LIN {X 0,Y 298.79,Z 342.264,A -85,B 0,C 180,E1 -16386.754,E2 -16386.754} C_VEL
LIN {X 0,Y 298.673,Z 342.283,A -85,B 0,C 180,E1 -16389.481,E2 -16389.481} C_VEL
LIN {X 0,Y 298.544,Z 342.297,A -85,B 0,C 180,E1 -16393.616,E2 -16393.616} C_VEL
LIN {X 0,Y 298.541,Z 342.295,A -85,B 0,C 180,E1 -16396.409,E2 -16396.409} C_VEL
LIN {X 0,Y 298.503,Z 342.301,A -85,B 0,C 180,E1 -16399.655,E2 -16399.655} C_VEL
LIN {X 0,Y 298.416,Z 342.312,A -85,B 0,C 180,E1 -16403.601,E2 -16403.601} C_VEL
LIN {X 0,Y 298.4,Z 342.315,A -85,B 0,C 180,E1 -16406.583,E2 -16406.583} C_VEL
LIN {X 0,Y 298.386,Z 342.315,A -85,B 0,C 180,E1 -16409.645,E2 -16409.645} C_VEL
LIN {X 0,Y 298.386,Z 342.319,A -85,B 0,C 180,E1 -16412.802,E2 -16412.802} C_VEL
LIN {X 0,Y 298.435,Z 342.313,A -85,B 0,C 180,E1 -16416.807,E2 -16416.807} C_VEL
LIN {X 0,Y 298.342,Z 342.321,A -85,B 0,C 180,E1 -16421.08,E2 -16421.08} C_VEL
LIN {X 0,Y 298.35,Z 342.321,A -85,B 0,C 180,E1 -16425.036,E2 -16425.036} C_VEL
LIN {X 0,Y 298.428,Z 342.312,A -85,B 0,C 180,E1 -16426.927,E2 -16426.927} C_VEL
LIN {X 0,Y 298.392,Z 342.316,A -85,B 0,C 180,E1 -16431.009,E2 -16431.009} C_VEL
LIN {X 0,Y 298.515,Z 343.786,A -85,B 0,C 180,E1 -16433.175,E2 -16433.175} C_VEL
LIN {X 0,Y 298.505,Z 345.953,A -85,B 0,C 180,E1 -16435.595,E2 -16435.595} C_VEL
LIN {X 0,Y 298.24,Z 348.977,A -85,B 0,C 180,E1 -16438.774,E2 -16438.774} C_VEL
LIN {X 0,Y 297.975,Z 352.015,A -85,B 0,C 180,E1 -16441.855,E2 -16441.855} C_VEL
LIN {X 0,Y 297.704,Z 355.744,A -85,B 0,C 180,E1 -16445.475,E2 -16445.475} C_VEL
LIN {X 0,Y 301.735,Z 369.34,A -85,B 0,C 180,E1 -16446.473,E2 -16446.473} C_VEL
LIN {X 0,Y 304.492,Z 381.011,A -85,B 0,C 180,E1 -16447.514,E2 -16447.514} C_VEL
LIN {X 0,Y 306.309,Z 391.773,A -85,B 0,C 180,E1 -16448.64,E2 -16448.64} C_VEL
LIN {X 0,Y 306.628,Z 395.068,A -85,B 0,C 180,E1 -16449.016,E2 -16449.016} C_VEL
LIN {X 0,Y 305.081,Z 406.409,A -85,B 0,C 180,E1 -16450.312,E2 -16450.312} C_VEL
LIN {X 0,Y 303.763,Z 416.336,A -85,B 0,C 180,E1 -16451.753,E2 -16451.753} C_VEL
LIN {X 0,Y 302.259,Z 425.786,A -85,B 0,C 180,E1 -16453.452,E2 -16453.452} C_VEL
LIN {X 0,Y 300.578,Z 434.694,A -85,B 0,C 180,E1 -16455.443,E2 -16455.443} C_VEL
LIN {X 0,Y 299.354,Z 441.858,A -85,B 0,C 180,E1 -16457.458,E2 -16457.458} C_VEL
LIN {X 0,Y 298.473,Z 446.69,A -85,B 0,C 180,E1 -16459.143,E2 -16459.143} C_VEL
LIN {X 0,Y 297.683,Z 451.382,A -85,B 0,C 180,E1 -16461.173,E2 -16461.173} C_VEL
LIN {X 0,Y 297.207,Z 455.108,A -85,B 0,C 180,E1 -16463.3,E2 -16463.3} C_VEL
LIN {X 0,Y 296.959,Z 456.824,A -85,B 0,C 180,E1 -16464.569,E2 -16464.569} C_VEL
LIN {X 0,Y 296.811,Z 458.217,A -85,B 0,C 180,E1 -16465.927,E2 -16465.927} C_VEL
LIN {X 0,Y 296.546,Z 459.821,A -85,B 0,C 180,E1 -16468.643,E2 -16468.643} C_VEL
LIN {X 0,Y 296.529,Z 460.051,A -85,B 0,C 180,E1 -16470.001,E2 -16470.001} C_VEL
LIN {X 0,Y 296.546,Z 459.859,A -85,B 0,C 180,E1 -16471.359,E2 -16471.359} C_VEL
LIN {X 0,Y 296.788,Z 458.304,A -85,B 0,C 180,E1 -16474.074,E2 -16474.074} C_VEL
LIN {X 0,Y 296.96,Z 456.948,A -85,B 0,C 180,E1 -16475.433,E2 -16475.433} C_VEL
LIN {X 0,Y 297.357,Z 454.082,A -85,B 0,C 180,E1 -16477.47,E2 -16477.47} C_VEL
LIN {X 0,Y 297.855,Z 450.199,A -85,B 0,C 180,E1 -16479.507,E2 -16479.507} C_VEL
LIN {X 0,Y 298.758,Z 445.181,A -85,B 0,C 180,E1 -16481.535,E2 -16481.535} C_VEL
LIN {X 0,Y 299.867,Z 438.863,A -85,B 0,C 180,E1 -16483.555,E2 -16483.555} C_VEL
LIN {X 0,Y 301.325,Z 430.953,A -85,B 0,C 180,E1 -16485.559,E2 -16485.559} C_VEL
LIN {X 0,Y 303.025,Z 421.112,A -85,B 0,C 180,E1 -16487.548,E2 -16487.548} C_VEL
LIN {X 0,Y 304.471,Z 410.784,A -85,B 0,C 180,E1 -16489.204,E2 -16489.204} C_VEL
LIN {X 0,Y 306.134,Z 399.125,A -85,B 0,C 180,E1 -16490.669,E2 -16490.669} C_VEL
LIN {X 0,Y 306.659,Z 394.489,A -85,B 0,C 180,E1 -16491.159,E2 -16491.159} C_VEL
LIN {X 0,Y 304.975,Z 383.491,A -85,B 0,C 180,E1 -16492.36,E2 -16492.36} C_VEL
LIN {X 0,Y 302.381,Z 371.646,A -85,B 0,C 180,E1 -16493.45,E2 -16493.45} C_VEL
LIN {X 0,Y 298.518,Z 358.662,A -85,B 0,C 180,E1 -16494.449,E2 -16494.449} C_VEL
LIN {X 0,Y 297.688,Z 355.729,A -85,B 0,C 180,E1 -16494.66,E2 -16494.66} C_VEL
LIN {X 0,Y 297.944,Z 352.136,A -85,B 0,C 180,E1 -16498.149,E2 -16498.149} C_VEL
LIN {X 0,Y 298.325,Z 348.377,A -85,B 0,C 180,E1 -16501.994,E2 -16501.994} C_VEL
LIN {X 0,Y 298.503,Z 345.997,A -85,B 0,C 180,E1 -16504.508,E2 -16504.508} C_VEL
LIN {X 0,Y 298.455,Z 343.087,A -85,B 0,C 180,E1 -16507.752,E2 -16507.752} C_VEL
LIN {X 0,Y 298.388,Z 342.318,A -85,B 0,C 180,E1 -16508.99,E2 -16508.99} C_VEL
LIN {X 0,Y 298.399,Z 342.317,A -85,B 0,C 180,E1 -16513.103,E2 -16513.103} C_VEL
LIN {X 0,Y 298.369,Z 342.319,A -85,B 0,C 180,E1 -16516.914,E2 -16516.914} C_VEL
LIN {X 0,Y 298.353,Z 342.32,A -85,B 0,C 180,E1 -16521.018,E2 -16521.018} C_VEL
LIN {X 0,Y 298.415,Z 342.312,A -85,B 0,C 180,E1 -16523.929,E2 -16523.929} C_VEL
LIN {X 0,Y 298.391,Z 342.318,A -85,B 0,C 180,E1 -16527.199,E2 -16527.199} C_VEL
LIN {X 0,Y 298.4,Z 342.314,A -85,B 0,C 180,E1 -16530.625,E2 -16530.625} C_VEL
LIN {X 0,Y 298.437,Z 342.31,A -85,B 0,C 180,E1 -16534.92,E2 -16534.92} C_VEL
LIN {X 0,Y 298.437,Z 342.31,A -85,B 0,C 180,E1 -16539.314,E2 -16539.314} C_VEL
LIN {X 0,Y 298.536,Z 342.296,A -85,B 0,C 180,E1 -16542.179,E2 -16542.179} C_VEL
LIN {X 0,Y 298.562,Z 342.293,A -85,B 0,C 180,E1 -16545.382,E2 -16545.382} C_VEL
LIN {X 0,Y 298.591,Z 342.29,A -85,B 0,C 180,E1 -16549.146,E2 -16549.146} C_VEL
LIN {X 0,Y 298.755,Z 342.269,A -85,B 0,C 180,E1 -16551.248,E2 -16551.248} C_VEL
LIN {X 0,Y 298.04,Z 342.361,A -85,B 0,C 180,E1 -16552.372,E2 -16552.372} C_VEL
LIN {X 0,Y 295.081,Z 342.728,A -85,B 0,C 180,E1 -16554.2,E2 -16554.2} C_VEL
LIN {X 0,Y 292.68,Z 343.025,A -85,B 0,C 180,E1 -16555.684,E2 -16555.684} C_VEL
LIN {X 0,Y 291.784,Z 343.139,A -85,B 0,C 180,E1 -16556.835,E2 -16556.835} C_VEL
LIN {X 0,Y 291.782,Z 343.137,A -85,B 0,C 180,E1 -16557.224,E2 -16557.224} C_VEL
LIN {X 0,Y 291.915,Z 343.123,A -85,B 0,C 180,E1 -16560,E2 -16560} C_VEL
LIN {X 0,Y 291.785,Z 343.138,A -85,B 0,C 180,E1 -16562.761,E2 -16562.761} C_VEL
LIN {X 0,Y 291.733,Z 343.144,A -85,B 0,C 180,E1 -16566.918,E2 -16566.918} C_VEL
LIN {X 0,Y 291.573,Z 343.166,A -85,B 0,C 180,E1 -16569.714,E2 -16569.714} C_VEL
LIN {X 0,Y 291.519,Z 343.175,A -85,B 0,C 180,E1 -16573.95,E2 -16573.95} C_VEL
LIN {X 0,Y 291.485,Z 343.175,A -85,B 0,C 180,E1 -16576.818,E2 -16576.818} C_VEL
LIN {X 0,Y 291.449,Z 343.183,A -85,B 0,C 180,E1 -16579.875,E2 -16579.875} C_VEL
LIN {X 0,Y 291.361,Z 343.191,A -85,B 0,C 180,E1 -16584.209,E2 -16584.209} C_VEL
LIN {X 0,Y 291.351,Z 343.194,A -85,B 0,C 180,E1 -16587.279,E2 -16587.279} C_VEL
LIN {X 0,Y 291.316,Z 343.197,A -85,B 0,C 180,E1 -16590.439,E2 -16590.439} C_VEL
LIN {X 0,Y 291.342,Z 343.197,A -85,B 0,C 180,E1 -16593.699,E2 -16593.699} C_VEL
LIN {X 0,Y 291.358,Z 343.195,A -85,B 0,C 180,E1 -16597.25,E2 -16597.25} C_VEL
LIN {X 0,Y 291.298,Z 343.198,A -85,B 0,C 180,E1 -16600.648,E2 -16600.648} C_VEL
LIN {X 0,Y 291.369,Z 343.359,A -85,B 0,C 180,E1 -16602.483,E2 -16602.483} C_VEL
LIN {X 0,Y 292.046,Z 347.294,A -85,B 0,C 180,E1 -16606.215,E2 -16606.215} C_VEL
LIN {X 0,Y 292.85,Z 351.787,A -85,B 0,C 180,E1 -16610.171,E2 -16610.171} C_VEL
LIN {X 0,Y 293.099,Z 355.448,A -85,B 0,C 180,E1 -16613.169,E2 -16613.169} C_VEL
LIN {X 0,Y 292.963,Z 358.663,A -85,B 0,C 180,E1 -16615.685,E2 -16615.685} C_VEL
LIN {X 0,Y 292.107,Z 364.486,A -85,B 0,C 180,E1 -16620.014,E2 -16620.014} C_VEL
LIN {X 0,Y 291.474,Z 368.769,A -85,B 0,C 180,E1 -16623.144,E2 -16623.144} C_VEL
LIN {X 0,Y 291.178,Z 371.049,A -85,B 0,C 180,E1 -16624.786,E2 -16624.786} C_VEL
LIN {X 0,Y 294.511,Z 384.98,A -85,B 0,C 180,E1 -16625.735,E2 -16625.735} C_VEL
LIN {X 0,Y 296.709,Z 397.246,A -85,B 0,C 180,E1 -16626.775,E2 -16626.775} C_VEL
LIN {X 0,Y 298.098,Z 409.454,A -85,B 0,C 180,E1 -16628.021,E2 -16628.021} C_VEL
LIN {X 0,Y 298.565,Z 417.315,A -85,B 0,C 180,E1 -16628.963,E2 -16628.963} C_VEL
LIN {X 0,Y 296.81,Z 428.854,A -85,B 0,C 180,E1 -16630.46,E2 -16630.46} C_VEL
LIN {X 0,Y 295.151,Z 439.157,A -85,B 0,C 180,E1 -16632.167,E2 -16632.167} C_VEL
LIN {X 0,Y 293.594,Z 448.125,A -85,B 0,C 180,E1 -16634.021,E2 -16634.021} C_VEL
LIN {X 0,Y 292.189,Z 456.149,A -85,B 0,C 180,E1 -16636.082,E2 -16636.082} C_VEL
LIN {X 0,Y 291.085,Z 462.584,A -85,B 0,C 180,E1 -16638.157,E2 -16638.157} C_VEL
LIN {X 0,Y 290.314,Z 467.698,A -85,B 0,C 180,E1 -16640.243,E2 -16640.243} C_VEL
LIN {X 0,Y 289.82,Z 471.673,A -85,B 0,C 180,E1 -16642.335,E2 -16642.335} C_VEL
LIN {X 0,Y 289.517,Z 474.61,A -85,B 0,C 180,E1 -16644.427,E2 -16644.427} C_VEL
LIN {X 0,Y 289.451,Z 476.01,A -85,B 0,C 180,E1 -16645.822,E2 -16645.822} C_VEL
LIN {X 0,Y 289.442,Z 477.01,A -85,B 0,C 180,E1 -16647.216,E2 -16647.216} C_VEL
LIN {X 0,Y 289.403,Z 477.619,A -85,B 0,C 180,E1 -16648.608,E2 -16648.608} C_VEL
LIN {X 0,Y 289.406,Z 477.834,A -85,B 0,C 180,E1 -16649.999,E2 -16649.999} C_VEL
LIN {X 0,Y 289.403,Z 477.615,A -85,B 0,C 180,E1 -16651.391,E2 -16651.391} C_VEL
LIN {X 0,Y 289.441,Z 477.004,A -85,B 0,C 180,E1 -16652.783,E2 -16652.783} C_VEL
LIN {X 0,Y 289.45,Z 476.002,A -85,B 0,C 180,E1 -16654.177,E2 -16654.177} C_VEL
LIN {X 0,Y 289.517,Z 474.598,A -85,B 0,C 180,E1 -16655.571,E2 -16655.571} C_VEL
LIN {X 0,Y 289.812,Z 471.652,A -85,B 0,C 180,E1 -16657.664,E2 -16657.664} C_VEL
LIN {X 0,Y 290.314,Z 467.667,A -85,B 0,C 180,E1 -16659.755,E2 -16659.755} C_VEL
LIN {X 0,Y 291.204,Z 461.543,A -85,B 0,C 180,E1 -16662.19,E2 -16662.19} C_VEL
LIN {X 0,Y 292.408,Z 454.86,A -85,B 0,C 180,E1 -16664.261,E2 -16664.261} C_VEL
LIN {X 0,Y 293.894,Z 446.57,A -85,B 0,C 180,E1 -16666.318,E2 -16666.318} C_VEL
LIN {X 0,Y 295.282,Z 438.07,A -85,B 0,C 180,E1 -16668.023,E2 -16668.023} C_VEL
LIN {X 0,Y 296.951,Z 427.571,A -85,B 0,C 180,E1 -16669.709,E2 -16669.709} C_VEL
LIN {X 0,Y 298.54,Z 417.189,A -85,B 0,C 180,E1 -16671.038,E2 -16671.038} C_VEL
LIN {X 0,Y 297.747,Z 405.797,A -85,B 0,C 180,E1 -16672.363,E2 -16672.363} C_VEL
LIN {X 0,Y 296.101,Z 393.226,A -85,B 0,C 180,E1 -16673.567,E2 -16673.567} C_VEL
LIN {X 0,Y 293.606,Z 380.807,A -85,B 0,C 180,E1 -16674.55,E2 -16674.55} C_VEL
LIN {X 0,Y 291.195,Z 371.057,A -85,B 0,C 180,E1 -16675.187,E2 -16675.187} C_VEL
LIN {X 0,Y 291.859,Z 366.099,A -85,B 0,C 180,E1 -16678.789,E2 -16678.789} C_VEL
LIN {X 0,Y 292.669,Z 360.646,A -85,B 0,C 180,E1 -16682.81,E2 -16682.81} C_VEL
LIN {X 0,Y 293.112,Z 357.233,A -85,B 0,C 180,E1 -16685.39,E2 -16685.39} C_VEL
LIN {X 0,Y 293.05,Z 353.256,A -85,B 0,C 180,E1 -16688.573,E2 -16688.573} C_VEL
LIN {X 0,Y 292.495,Z 349.393,A -85,B 0,C 180,E1 -16691.853,E2 -16691.853} C_VEL
LIN {X 0,Y 291.72,Z 345.229,A -85,B 0,C 180,E1 -16695.681,E2 -16695.681} C_VEL
LIN {X 0,Y 291.343,Z 343.196,A -85,B 0,C 180,E1 -16697.767,E2 -16697.767} C_VEL
LIN {X 0,Y 291.328,Z 343.199,A -85,B 0,C 180,E1 -16701.154,E2 -16701.154} C_VEL
LIN {X 0,Y 291.349,Z 343.196,A -85,B 0,C 180,E1 -16704.624,E2 -16704.624} C_VEL
LIN {X 0,Y 291.359,Z 343.192,A -85,B 0,C 180,E1 -16707.949,E2 -16707.949} C_VEL
LIN {X 0,Y 291.336,Z 343.195,A -85,B 0,C 180,E1 -16711.153,E2 -16711.153} C_VEL
LIN {X 0,Y 291.354,Z 343.195,A -85,B 0,C 180,E1 -16714.266,E2 -16714.266} C_VEL
LIN {X 0,Y 291.365,Z 343.19,A -85,B 0,C 180,E1 -16717.298,E2 -16717.298} C_VEL
LIN {X 0,Y 291.451,Z 343.182,A -85,B 0,C 180,E1 -16720.27,E2 -16720.27} C_VEL
LIN {X 0,Y 291.533,Z 343.17,A -85,B 0,C 180,E1 -16724.634,E2 -16724.634} C_VEL
LIN {X 0,Y 291.528,Z 343.168,A -85,B 0,C 180,E1 -16728.88,E2 -16728.88} C_VEL
LIN {X 0,Y 291.702,Z 343.15,A -85,B 0,C 180,E1 -16731.688,E2 -16731.688} C_VEL
LIN {X 0,Y 291.625,Z 343.157,A -85,B 0,C 180,E1 -16734.468,E2 -16734.468} C_VEL
LIN {X 0,Y 291.876,Z 343.125,A -85,B 0,C 180,E1 -16738.62,E2 -16738.62} C_VEL
LIN {X 0,Y 291.876,Z 343.128,A -85,B 0,C 180,E1 -16741.38,E2 -16741.38} C_VEL
LIN {X 0,Y 291.739,Z 343.143,A -85,B 0,C 180,E1 -16746.918,E2 -16746.918} C_VEL
LIN {X 0,Y 291.621,Z 343.16,A -85,B 0,C 180,E1 -16749.712,E2 -16749.712} C_VEL
LIN {X 0,Y 291.514,Z 343.17,A -85,B 0,C 180,E1 -16753.951,E2 -16753.951} C_VEL
LIN {X 0,Y 291.479,Z 343.176,A -85,B 0,C 180,E1 -16756.818,E2 -16756.818} C_VEL
LIN {X 0,Y 291.444,Z 343.179,A -85,B 0,C 180,E1 -16759.875,E2 -16759.875} C_VEL
LIN {X 0,Y 291.356,Z 343.19,A -85,B 0,C 180,E1 -16764.209,E2 -16764.209} C_VEL
LIN {X 0,Y 291.346,Z 343.194,A -85,B 0,C 180,E1 -16767.279,E2 -16767.279} C_VEL
LIN {X 0,Y 291.312,Z 343.198,A -85,B 0,C 180,E1 -16770.44,E2 -16770.44} C_VEL
LIN {X 0,Y 291.337,Z 343.193,A -85,B 0,C 180,E1 -16773.7,E2 -16773.7} C_VEL
LIN {X 0,Y 291.362,Z 343.191,A -85,B 0,C 180,E1 -16777.253,E2 -16777.253} C_VEL
LIN {X 0,Y 291.294,Z 343.201,A -85,B 0,C 180,E1 -16780.649,E2 -16780.649} C_VEL
LIN {X 0,Y 291.278,Z 343.204,A -85,B 0,C 180,E1 -16784.405,E2 -16784.405} C_VEL
LIN {X 0,Y 291.352,Z 343.195,A -85,B 0,C 180,E1 -16788.399,E2 -16788.399} C_VEL
LIN {X 0,Y 291.335,Z 343.195,A -85,B 0,C 180,E1 -16791.157,E2 -16791.157} C_VEL
LIN {X 0,Y 291.471,Z 344.663,A -85,B 0,C 180,E1 -16792.931,E2 -16792.931} C_VEL
LIN {X 0,Y 291.403,Z 347.671,A -85,B 0,C 180,E1 -16796.311,E2 -16796.311} C_VEL
LIN {X 0,Y 291.113,Z 350.699,A -85,B 0,C 180,E1 -16799.539,E2 -16799.539} C_VEL
LIN {X 0,Y 290.796,Z 354.517,A -85,B 0,C 180,E1 -16803.409,E2 -16803.409} C_VEL
LIN {X 0,Y 290.677,Z 355.97,A -85,B 0,C 180,E1 -16804.836,E2 -16804.836} C_VEL
LIN {X 0,Y 294.851,Z 369.828,A -85,B 0,C 180,E1 -16805.905,E2 -16805.905} C_VEL
LIN {X 0,Y 297.743,Z 381.66,A -85,B 0,C 180,E1 -16807.009,E2 -16807.009} C_VEL
LIN {X 0,Y 299.48,Z 392.003,A -85,B 0,C 180,E1 -16808.128,E2 -16808.128} C_VEL
LIN {X 0,Y 299.824,Z 396.866,A -85,B 0,C 180,E1 -16808.696,E2 -16808.696} C_VEL
LIN {X 0,Y 298.24,Z 407.907,A -85,B 0,C 180,E1 -16810.021,E2 -16810.021} C_VEL
LIN {X 0,Y 296.925,Z 417.177,A -85,B 0,C 180,E1 -16811.427,E2 -16811.427} C_VEL
LIN {X 0,Y 295.447,Z 426.004,A -85,B 0,C 180,E1 -16813.059,E2 -16813.059} C_VEL
LIN {X 0,Y 293.718,Z 434.912,A -85,B 0,C 180,E1 -16815.096,E2 -16815.096} C_VEL
LIN {X 0,Y 292.423,Z 442.076,A -85,B 0,C 180,E1 -16817.156,E2 -16817.156} C_VEL
LIN {X 0,Y 291.503,Z 446.907,A -85,B 0,C 180,E1 -16818.88,E2 -16818.88} C_VEL
LIN {X 0,Y 290.662,Z 451.599,A -85,B 0,C 180,E1 -16820.958,E2 -16820.958} C_VEL
LIN {X 0,Y 290.119,Z 455.604,A -85,B 0,C 180,E1 -16823.32,E2 -16823.32} C_VEL
LIN {X 0,Y 289.73,Z 458.433,A -85,B 0,C 180,E1 -16825.828,E2 -16825.828} C_VEL
LIN {X 0,Y 289.467,Z 460.036,A -85,B 0,C 180,E1 -16828.609,E2 -16828.609} C_VEL
LIN {X 0,Y 289.446,Z 460.266,A -85,B 0,C 180,E1 -16830.001,E2 -16830.001} C_VEL
LIN {X 0,Y 289.467,Z 460.073,A -85,B 0,C 180,E1 -16831.392,E2 -16831.392} C_VEL
LIN {X 0,Y 289.709,Z 458.519,A -85,B 0,C 180,E1 -16834.174,E2 -16834.174} C_VEL
LIN {X 0,Y 290.119,Z 455.759,A -85,B 0,C 180,E1 -16836.679,E2 -16836.679} C_VEL
LIN {X 0,Y 290.628,Z 451.826,A -85,B 0,C 180,E1 -16839.044,E2 -16839.044} C_VEL
LIN {X 0,Y 291.469,Z 447.193,A -85,B 0,C 180,E1 -16841.122,E2 -16841.122} C_VEL
LIN {X 0,Y 292.784,Z 440.208,A -85,B 0,C 180,E1 -16843.535,E2 -16843.535} C_VEL
LIN {X 0,Y 294.202,Z 432.635,A -85,B 0,C 180,E1 -16845.59,E2 -16845.59} C_VEL
LIN {X 0,Y 295.669,Z 424.872,A -85,B 0,C 180,E1 -16847.285,E2 -16847.285} C_VEL
LIN {X 0,Y 297.171,Z 414.978,A -85,B 0,C 180,E1 -16849.046,E2 -16849.046} C_VEL
LIN {X 0,Y 298.693,Z 404.861,A -85,B 0,C 180,E1 -16850.487,E2 -16850.487} C_VEL
LIN {X 0,Y 299.887,Z 396.275,A -85,B 0,C 180,E1 -16851.48,E2 -16851.48} C_VEL
LIN {X 0,Y 298.597,Z 386.445,A -85,B 0,C 180,E1 -16852.61,E2 -16852.61} C_VEL
LIN {X 0,Y 296.355,Z 375.616,A -85,B 0,C 180,E1 -16853.695,E2 -16853.695} C_VEL
LIN {X 0,Y 293.032,Z 363.689,A -85,B 0,C 180,E1 -16854.718,E2 -16854.718} C_VEL
LIN {X 0,Y 290.678,Z 355.979,A -85,B 0,C 180,E1 -16855.275,E2 -16855.275} C_VEL
LIN {X 0,Y 291.081,Z 351.622,A -85,B 0,C 180,E1 -16859.633,E2 -16859.633} C_VEL
LIN {X 0,Y 291.336,Z 349.015,A -85,B 0,C 180,E1 -16862.401,E2 -16862.401} C_VEL
LIN {X 0,Y 291.493,Z 346.287,A -85,B 0,C 180,E1 -16865.355,E2 -16865.355} C_VEL
LIN {X 0,Y 291.489,Z 344.587,A -85,B 0,C 180,E1 -16867.283,E2 -16867.283} C_VEL
LIN {X 0,Y 291.343,Z 343.282,A -85,B 0,C 180,E1 -16868.843,E2 -16868.843} C_VEL
LIN {X 0,Y 291.32,Z 343.198,A -85,B 0,C 180,E1 -16872.492,E2 -16872.492} C_VEL
LIN {X 0,Y 291.288,Z 343.201,A -85,B 0,C 180,E1 -16876.37,E2 -16876.37} C_VEL
LIN {X 0,Y 291.311,Z 343.196,A -85,B 0,C 180,E1 -16880.535,E2 -16880.535} C_VEL
LIN {X 0,Y 291.397,Z 343.187,A -85,B 0,C 180,E1 -16882.918,E2 -16882.918} C_VEL
LIN {X 0,Y 291.343,Z 343.192,A -85,B 0,C 180,E1 -16886.301,E2 -16886.301} C_VEL
LIN {X 0,Y 291.363,Z 343.189,A -85,B 0,C 180,E1 -16890.268,E2 -16890.268} C_VEL
LIN {X 0,Y 291.357,Z 343.19,A -85,B 0,C 180,E1 -16894.266,E2 -16894.266} C_VEL
LIN {X 0,Y 291.37,Z 343.19,A -85,B 0,C 180,E1 -16897.298,E2 -16897.298} C_VEL
LIN {X 0,Y 291.457,Z 343.178,A -85,B 0,C 180,E1 -16900.27,E2 -16900.27} C_VEL
LIN {X 0,Y 291.554,Z 343.169,A -85,B 0,C 180,E1 -16904.623,E2 -16904.623} C_VEL
LIN {X 0,Y 291.534,Z 343.171,A -85,B 0,C 180,E1 -16908.88,E2 -16908.88} C_VEL
LIN {X 0,Y 291.708,Z 343.146,A -85,B 0,C 180,E1 -16911.688,E2 -16911.688} C_VEL
LIN {X 0,Y 291.628,Z 343.161,A -85,B 0,C 180,E1 -16914.468,E2 -16914.468} C_VEL
LIN {X 0,Y 291.782,Z 343.137,A -85,B 0,C 180,E1 -16917.224,E2 -16917.224} C_VEL
LIN {X 0,Y 291.317,Z 343.201,A -85,B 0,C 180,E1 -16918.377,E2 -16918.377} C_VEL
LIN {X 0,Y 289.82,Z 343.389,A -85,B 0,C 180,E1 -16919.509,E2 -16919.509} C_VEL
LIN {X 0,Y 285.991,Z 343.861,A -85,B 0,C 180,E1 -16921.778,E2 -16921.778} C_VEL
LIN {X 0,Y 284.782,Z 344.01,A -85,B 0,C 180,E1 -16922.96,E2 -16922.96} C_VEL
LIN {X 0,Y 284.63,Z 344.028,A -85,B 0,C 180,E1 -16923.362,E2 -16923.362} C_VEL
LIN {X 0,Y 284.685,Z 344.022,A -85,B 0,C 180,E1 -16927.09,E2 -16927.09} C_VEL
LIN {X 0,Y 284.517,Z 344.047,A -85,B 0,C 180,E1 -16929.957,E2 -16929.957} C_VEL
LIN {X 0,Y 284.476,Z 344.051,A -85,B 0,C 180,E1 -16934.303,E2 -16934.303} C_VEL
LIN {X 0,Y 284.423,Z 344.056,A -85,B 0,C 180,E1 -16937.248,E2 -16937.248} C_VEL
LIN {X 0,Y 284.376,Z 344.062,A -85,B 0,C 180,E1 -16940.242,E2 -16940.242} C_VEL
LIN {X 0,Y 284.321,Z 344.07,A -85,B 0,C 180,E1 -16943.854,E2 -16943.854} C_VEL
LIN {X 0,Y 284.281,Z 344.075,A -85,B 0,C 180,E1 -16948.016,E2 -16948.016} C_VEL
LIN {X 0,Y 284.283,Z 344.076,A -85,B 0,C 180,E1 -16951.276,E2 -16951.276} C_VEL
LIN {X 0,Y 284.335,Z 344.07,A -85,B 0,C 180,E1 -16955.347,E2 -16955.347} C_VEL
LIN {X 0,Y 284.297,Z 344.072,A -85,B 0,C 180,E1 -16958.172,E2 -16958.172} C_VEL
LIN {X 0,Y 284.277,Z 344.153,A -85,B 0,C 180,E1 -16961.875,E2 -16961.875} C_VEL
LIN {X 0,Y 284.955,Z 348.026,A -85,B 0,C 180,E1 -16965.663,E2 -16965.663} C_VEL
LIN {X 0,Y 285.776,Z 352.392,A -85,B 0,C 180,E1 -16969.674,E2 -16969.674} C_VEL
LIN {X 0,Y 286.075,Z 356.323,A -85,B 0,C 180,E1 -16972.995,E2 -16972.995} C_VEL
LIN {X 0,Y 285.965,Z 359.535,A -85,B 0,C 180,E1 -16975.58,E2 -16975.58} C_VEL
LIN {X 0,Y 285.134,Z 364.816,A -85,B 0,C 180,E1 -16979.619,E2 -16979.619} C_VEL
LIN {X 0,Y 284.309,Z 370.096,A -85,B 0,C 180,E1 -16983.58,E2 -16983.58} C_VEL
LIN {X 0,Y 284.224,Z 370.828,A -85,B 0,C 180,E1 -16984.125,E2 -16984.125} C_VEL
LIN {X 0,Y 287.574,Z 384.322,A -85,B 0,C 180,E1 -16985.083,E2 -16985.083} C_VEL
LIN {X 0,Y 289.892,Z 397.148,A -85,B 0,C 180,E1 -16986.205,E2 -16986.205} C_VEL
LIN {X 0,Y 291.273,Z 409.236,A -85,B 0,C 180,E1 -16987.478,E2 -16987.478} C_VEL
LIN {X 0,Y 291.737,Z 418.533,A -85,B 0,C 180,E1 -16988.631,E2 -16988.631} C_VEL
LIN {X 0,Y 289.924,Z 429.774,A -85,B 0,C 180,E1 -16990.161,E2 -16990.161} C_VEL
LIN {X 0,Y 288.306,Z 439.314,A -85,B 0,C 180,E1 -16991.805,E2 -16991.805} C_VEL
LIN {X 0,Y 286.757,Z 447.911,A -85,B 0,C 180,E1 -16993.629,E2 -16993.629} C_VEL
LIN {X 0,Y 285.269,Z 455.934,A -85,B 0,C 180,E1 -16995.737,E2 -16995.737} C_VEL
LIN {X 0,Y 284.091,Z 462.368,A -85,B 0,C 180,E1 -16997.861,E2 -16997.861} C_VEL
LIN {X 0,Y 283.276,Z 467.482,A -85,B 0,C 180,E1 -16999.998,E2 -16999.998} C_VEL
LIN {X 0,Y 282.754,Z 471.457,A -85,B 0,C 180,E1 -17002.142,E2 -17002.142} C_VEL
LIN {X 0,Y 282.411,Z 474.64,A -85,B 0,C 180,E1 -17004.521,E2 -17004.521} C_VEL
LIN {X 0,Y 282.35,Z 476.795,A -85,B 0,C 180,E1 -17007.146,E2 -17007.146} C_VEL
LIN {X 0,Y 282.327,Z 477.404,A -85,B 0,C 180,E1 -17008.573,E2 -17008.573} C_VEL
LIN {X 0,Y 282.328,Z 477.62,A -85,B 0,C 180,E1 -17009.999,E2 -17009.999} C_VEL
LIN {X 0,Y 282.327,Z 477.4,A -85,B 0,C 180,E1 -17011.426,E2 -17011.426} C_VEL
LIN {X 0,Y 282.349,Z 476.788,A -85,B 0,C 180,E1 -17012.853,E2 -17012.853} C_VEL
LIN {X 0,Y 282.41,Z 474.628,A -85,B 0,C 180,E1 -17015.477,E2 -17015.477} C_VEL
LIN {X 0,Y 282.747,Z 471.435,A -85,B 0,C 180,E1 -17017.857,E2 -17017.857} C_VEL
LIN {X 0,Y 283.276,Z 467.449,A -85,B 0,C 180,E1 -17020,E2 -17020} C_VEL
LIN {X 0,Y 284.229,Z 461.325,A -85,B 0,C 180,E1 -17022.494,E2 -17022.494} C_VEL
LIN {X 0,Y 285.506,Z 454.641,A -85,B 0,C 180,E1 -17024.614,E2 -17024.614} C_VEL
LIN {X 0,Y 287.075,Z 446.352,A -85,B 0,C 180,E1 -17026.717,E2 -17026.717} C_VEL
LIN {X 0,Y 288.502,Z 437.85,A -85,B 0,C 180,E1 -17028.461,E2 -17028.461} C_VEL
LIN {X 0,Y 290.26,Z 427.352,A -85,B 0,C 180,E1 -17030.183,E2 -17030.183} C_VEL
LIN {X 0,Y 291.727,Z 418.398,A -85,B 0,C 180,E1 -17031.368,E2 -17031.368} C_VEL
LIN {X 0,Y 291.061,Z 407.28,A -85,B 0,C 180,E1 -17032.726,E2 -17032.726} C_VEL
LIN {X 0,Y 289.483,Z 394.534,A -85,B 0,C 180,E1 -17034.026,E2 -17034.026} C_VEL
LIN {X 0,Y 286.949,Z 381.735,A -85,B 0,C 180,E1 -17035.097,E2 -17035.097} C_VEL
LIN {X 0,Y 284.226,Z 370.799,A -85,B 0,C 180,E1 -17035.875,E2 -17035.875} C_VEL
LIN {X 0,Y 284.942,Z 365.886,A -85,B 0,C 180,E1 -17039.556,E2 -17039.556} C_VEL
LIN {X 0,Y 285.713,Z 361.03,A -85,B 0,C 180,E1 -17043.245,E2 -17043.245} C_VEL
LIN {X 0,Y 286.076,Z 357.364,A -85,B 0,C 180,E1 -17046.127,E2 -17046.127} C_VEL
LIN {X 0,Y 286.066,Z 354.879,A -85,B 0,C 180,E1 -17048.171,E2 -17048.171} C_VEL
LIN {X 0,Y 285.808,Z 352.343,A -85,B 0,C 180,E1 -17050.333,E2 -17050.333} C_VEL
LIN {X 0,Y 285.014,Z 347.953,A -85,B 0,C 180,E1 -17054.349,E2 -17054.349} C_VEL
LIN {X 0,Y 284.272,Z 344.077,A -85,B 0,C 180,E1 -17058.243,E2 -17058.243} C_VEL
LIN {X 0,Y 284.303,Z 344.072,A -85,B 0,C 180,E1 -17062.281,E2 -17062.281} C_VEL
LIN {X 0,Y 284.301,Z 344.071,A -85,B 0,C 180,E1 -17065.35,E2 -17065.35} C_VEL
LIN {X 0,Y 284.278,Z 344.076,A -85,B 0,C 180,E1 -17068.723,E2 -17068.723} C_VEL
LIN {X 0,Y 284.276,Z 344.075,A -85,B 0,C 180,E1 -17071.983,E2 -17071.983} C_VEL
LIN {X 0,Y 284.316,Z 344.071,A -85,B 0,C 180,E1 -17076.145,E2 -17076.145} C_VEL
LIN {X 0,Y 284.38,Z 344.062,A -85,B 0,C 180,E1 -17079.897,E2 -17079.897} C_VEL
LIN {X 0,Y 284.471,Z 344.05,A -85,B 0,C 180,E1 -17084.469,E2 -17084.469} C_VEL
LIN {X 0,Y 284.48,Z 344.047,A -85,B 0,C 180,E1 -17088.601,E2 -17088.601} C_VEL
LIN {X 0,Y 284.652,Z 344.027,A -85,B 0,C 180,E1 -17091.481,E2 -17091.481} C_VEL
LIN {X 0,Y 284.596,Z 344.034,A -85,B 0,C 180,E1 -17094.331,E2 -17094.331} C_VEL
LIN {X 0,Y 284.843,Z 344.002,A -85,B 0,C 180,E1 -17098.586,E2 -17098.586} C_VEL
LIN {X 0,Y 284.842,Z 344.005,A -85,B 0,C 180,E1 -17101.414,E2 -17101.414} C_VEL
LIN {X 0,Y 284.691,Z 344.022,A -85,B 0,C 180,E1 -17107.09,E2 -17107.09} C_VEL
LIN {X 0,Y 284.559,Z 344.038,A -85,B 0,C 180,E1 -17109.956,E2 -17109.956} C_VEL
LIN {X 0,Y 284.474,Z 344.046,A -85,B 0,C 180,E1 -17114.303,E2 -17114.303} C_VEL
LIN {X 0,Y 284.418,Z 344.058,A -85,B 0,C 180,E1 -17117.249,E2 -17117.249} C_VEL
LIN {X 0,Y 284.371,Z 344.06,A -85,B 0,C 180,E1 -17120.243,E2 -17120.243} C_VEL
LIN {X 0,Y 284.317,Z 344.067,A -85,B 0,C 180,E1 -17123.855,E2 -17123.855} C_VEL
LIN {X 0,Y 284.276,Z 344.072,A -85,B 0,C 180,E1 -17128.017,E2 -17128.017} C_VEL
LIN {X 0,Y 284.278,Z 344.074,A -85,B 0,C 180,E1 -17131.277,E2 -17131.277} C_VEL
LIN {X 0,Y 284.331,Z 344.067,A -85,B 0,C 180,E1 -17135.348,E2 -17135.348} C_VEL
LIN {X 0,Y 284.295,Z 344.071,A -85,B 0,C 180,E1 -17138.172,E2 -17138.172} C_VEL
LIN {X 0,Y 284.232,Z 344.079,A -85,B 0,C 180,E1 -17142.118,E2 -17142.118} C_VEL
LIN {X 0,Y 284.269,Z 344.077,A -85,B 0,C 180,E1 -17146.194,E2 -17146.194} C_VEL
LIN {X 0,Y 284.304,Z 344.073,A -85,B 0,C 180,E1 -17150.025,E2 -17150.025} C_VEL
LIN {X 0,Y 284.416,Z 345.205,A -85,B 0,C 180,E1 -17152.254,E2 -17152.254} C_VEL
LIN {X 0,Y 284.428,Z 347.879,A -85,B 0,C 180,E1 -17155.369,E2 -17155.369} C_VEL
LIN {X 0,Y 284.15,Z 350.916,A -85,B 0,C 180,E1 -17158.709,E2 -17158.709} C_VEL
LIN {X 0,Y 283.849,Z 354.002,A -85,B 0,C 180,E1 -17161.939,E2 -17161.939} C_VEL
LIN {X 0,Y 283.698,Z 356.198,A -85,B 0,C 180,E1 -17164.179,E2 -17164.179} C_VEL
LIN {X 0,Y 286.059,Z 363.77,A -85,B 0,C 180,E1 -17164.749,E2 -17164.749} C_VEL
LIN {X 0,Y 289.579,Z 376.233,A -85,B 0,C 180,E1 -17165.863,E2 -17165.863} C_VEL
LIN {X 0,Y 291.873,Z 387.392,A -85,B 0,C 180,E1 -17167.025,E2 -17167.025} C_VEL
LIN {X 0,Y 293.182,Z 397.088,A -85,B 0,C 180,E1 -17168.189,E2 -17168.189} C_VEL
LIN {X 0,Y 291.575,Z 408.127,A -85,B 0,C 180,E1 -17169.544,E2 -17169.544} C_VEL
LIN {X 0,Y 290.104,Z 417.971,A -85,B 0,C 180,E1 -17171.081,E2 -17171.081} C_VEL
LIN {X 0,Y 288.351,Z 427.843,A -85,B 0,C 180,E1 -17172.995,E2 -17172.995} C_VEL
LIN {X 0,Y 286.609,Z 436.457,A -85,B 0,C 180,E1 -17175.081,E2 -17175.081} C_VEL
LIN {X 0,Y 285.283,Z 443.321,A -85,B 0,C 180,E1 -17177.191,E2 -17177.191} C_VEL
LIN {X 0,Y 284.199,Z 448.815,A -85,B 0,C 180,E1 -17179.312,E2 -17179.312} C_VEL
LIN {X 0,Y 283.41,Z 453.126,A -85,B 0,C 180,E1 -17181.444,E2 -17181.444} C_VEL
LIN {X 0,Y 283.023,Z 456.087,A -85,B 0,C 180,E1 -17183.354,E2 -17183.354} C_VEL
LIN {X 0,Y 282.653,Z 458.649,A -85,B 0,C 180,E1 -17185.723,E2 -17185.723} C_VEL
LIN {X 0,Y 282.39,Z 460.251,A -85,B 0,C 180,E1 -17188.575,E2 -17188.575} C_VEL
LIN {X 0,Y 282.366,Z 460.481,A -85,B 0,C 180,E1 -17190.001,E2 -17190.001} C_VEL
LIN {X 0,Y 282.39,Z 460.288,A -85,B 0,C 180,E1 -17191.427,E2 -17191.427} C_VEL
LIN {X 0,Y 282.494,Z 459.701,A -85,B 0,C 180,E1 -17192.853,E2 -17192.853} C_VEL
LIN {X 0,Y 282.634,Z 458.734,A -85,B 0,C 180,E1 -17194.279,E2 -17194.279} C_VEL
LIN {X 0,Y 283.016,Z 456.242,A -85,B 0,C 180,E1 -17196.632,E2 -17196.632} C_VEL
LIN {X 0,Y 283.613,Z 452.04,A -85,B 0,C 180,E1 -17199.27,E2 -17199.27} C_VEL
LIN {X 0,Y 284.509,Z 447.406,A -85,B 0,C 180,E1 -17201.398,E2 -17201.398} C_VEL
LIN {X 0,Y 285.852,Z 440.422,A -85,B 0,C 180,E1 -17203.87,E2 -17203.87} C_VEL
LIN {X 0,Y 287.383,Z 432.848,A -85,B 0,C 180,E1 -17205.97,E2 -17205.97} C_VEL
LIN {X 0,Y 288.907,Z 425.084,A -85,B 0,C 180,E1 -17207.703,E2 -17207.703} C_VEL
LIN {X 0,Y 290.426,Z 415.525,A -85,B 0,C 180,E1 -17209.449,E2 -17209.449} C_VEL
LIN {X 0,Y 292.054,Z 405.071,A -85,B 0,C 180,E1 -17210.975,E2 -17210.975} C_VEL
LIN {X 0,Y 293.162,Z 396.488,A -85,B 0,C 180,E1 -17211.999,E2 -17211.999} C_VEL
LIN {X 0,Y 291.522,Z 385.309,A -85,B 0,C 180,E1 -17213.32,E2 -17213.32} C_VEL
LIN {X 0,Y 288.833,Z 373.401,A -85,B 0,C 180,E1 -17214.533,E2 -17214.533} C_VEL
LIN {X 0,Y 285.322,Z 361.51,A -85,B 0,C 180,E1 -17215.555,E2 -17215.555} C_VEL
LIN {X 0,Y 283.703,Z 356.177,A -85,B 0,C 180,E1 -17215.964,E2 -17215.964} C_VEL
LIN {X 0,Y 284.062,Z 352.236,A -85,B 0,C 180,E1 -17220.01,E2 -17220.01} C_VEL
LIN {X 0,Y 284.318,Z 349.531,A -85,B 0,C 180,E1 -17222.944,E2 -17222.944} C_VEL
LIN {X 0,Y 284.46,Z 346.504,A -85,B 0,C 180,E1 -17226.367,E2 -17226.367} C_VEL
LIN {X 0,Y 284.385,Z 344.979,A -85,B 0,C 180,E1 -17228.157,E2 -17228.157} C_VEL
LIN {X 0,Y 284.306,Z 344.073,A -85,B 0,C 180,E1 -17229.995,E2 -17229.995} C_VEL
LIN {X 0,Y 284.246,Z 344.08,A -85,B 0,C 180,E1 -17234.19,E2 -17234.19} C_VEL
LIN {X 0,Y 284.238,Z 344.078,A -85,B 0,C 180,E1 -17238.118,E2 -17238.118} C_VEL
LIN {X 0,Y 284.306,Z 344.069,A -85,B 0,C 180,E1 -17242.282,E2 -17242.282} C_VEL
LIN {X 0,Y 284.308,Z 344.071,A -85,B 0,C 180,E1 -17245.35,E2 -17245.35} C_VEL
LIN {X 0,Y 284.284,Z 344.071,A -85,B 0,C 180,E1 -17248.724,E2 -17248.724} C_VEL
LIN {X 0,Y 284.282,Z 344.071,A -85,B 0,C 180,E1 -17251.984,E2 -17251.984} C_VEL
LIN {X 0,Y 284.319,Z 344.066,A -85,B 0,C 180,E1 -17256.147,E2 -17256.147} C_VEL
LIN {X 0,Y 284.386,Z 344.058,A -85,B 0,C 180,E1 -17259.898,E2 -17259.898} C_VEL
LIN {X 0,Y 284.491,Z 344.048,A -85,B 0,C 180,E1 -17264.459,E2 -17264.459} C_VEL
LIN {X 0,Y 284.486,Z 344.049,A -85,B 0,C 180,E1 -17268.601,E2 -17268.601} C_VEL
LIN {X 0,Y 284.658,Z 344.025,A -85,B 0,C 180,E1 -17271.481,E2 -17271.481} C_VEL
LIN {X 0,Y 284.599,Z 344.035,A -85,B 0,C 180,E1 -17274.331,E2 -17274.331} C_VEL
LIN {X 0,Y 284.848,Z 344.004,A -85,B 0,C 180,E1 -17278.586,E2 -17278.586} C_VEL
LIN {X 0,Y 284.847,Z 344,A -85,B 0,C 180,E1 -17281.414,E2 -17281.414} C_VEL
LIN {X 0,Y 284.63,Z 344.028,A -85,B 0,C 180,E1 -17283.362,E2 -17283.362} C_VEL
LIN {X 0,Y 283.839,Z 344.13,A -85,B 0,C 180,E1 -17284.543,E2 -17284.543} C_VEL
LIN {X 0,Y 281.009,Z 344.483,A -85,B 0,C 180,E1 -17286.471,E2 -17286.471} C_VEL
LIN {X 0,Y 278.659,Z 344.777,A -85,B 0,C 180,E1 -17288.035,E2 -17288.035} C_VEL
LIN {X 0,Y 277.499,Z 344.917,A -85,B 0,C 180,E1 -17289.655,E2 -17289.655} C_VEL
LIN {X 0,Y 277.414,Z 344.929,A -85,B 0,C 180,E1 -17293.18,E2 -17293.18} C_VEL
LIN {X 0,Y 277.4,Z 344.933,A -85,B 0,C 180,E1 -17296.182,E2 -17296.182} C_VEL
LIN {X 0,Y 277.343,Z 344.938,A -85,B 0,C 180,E1 -17300.349,E2 -17300.349} C_VEL
LIN {X 0,Y 277.277,Z 344.946,A -85,B 0,C 180,E1 -17304.152,E2 -17304.152} C_VEL
LIN {X 0,Y 277.268,Z 344.949,A -85,B 0,C 180,E1 -17307.483,E2 -17307.483} C_VEL
LIN {X 0,Y 277.247,Z 344.95,A -85,B 0,C 180,E1 -17310.473,E2 -17310.473} C_VEL
LIN {X 0,Y 277.244,Z 344.953,A -85,B 0,C 180,E1 -17313.896,E2 -17313.896} C_VEL
LIN {X 0,Y 277.254,Z 344.951,A -85,B 0,C 180,E1 -17317.472,E2 -17317.472} C_VEL
LIN {X 0,Y 277.273,Z 345.163,A -85,B 0,C 180,E1 -17321.467,E2 -17321.467} C_VEL
LIN {X 0,Y 277.861,Z 348.721,A -85,B 0,C 180,E1 -17325.09,E2 -17325.09} C_VEL
LIN {X 0,Y 278.668,Z 353.035,A -85,B 0,C 180,E1 -17329.165,E2 -17329.165} C_VEL
LIN {X 0,Y 279.059,Z 357.186,A -85,B 0,C 180,E1 -17332.812,E2 -17332.812} C_VEL
LIN {X 0,Y 278.957,Z 360.398,A -85,B 0,C 180,E1 -17335.469,E2 -17335.469} C_VEL
LIN {X 0,Y 278.076,Z 365.702,A -85,B 0,C 180,E1 -17339.637,E2 -17339.637} C_VEL
LIN {X 0,Y 277.289,Z 370.622,A -85,B 0,C 180,E1 -17343.431,E2 -17343.431} C_VEL
LIN {X 0,Y 280.683,Z 384.263,A -85,B 0,C 180,E1 -17344.438,E2 -17344.438} C_VEL
LIN {X 0,Y 282.987,Z 396.438,A -85,B 0,C 180,E1 -17345.545,E2 -17345.545} C_VEL
LIN {X 0,Y 284.427,Z 408.63,A -85,B 0,C 180,E1 -17346.863,E2 -17346.863} C_VEL
LIN {X 0,Y 285.01,Z 418.351,A -85,B 0,C 180,E1 -17348.106,E2 -17348.106} C_VEL
LIN {X 0,Y 283.241,Z 429.561,A -85,B 0,C 180,E1 -17349.673,E2 -17349.673} C_VEL
LIN {X 0,Y 281.552,Z 439.006,A -85,B 0,C 180,E1 -17351.333,E2 -17351.333} C_VEL
LIN {X 0,Y 279.943,Z 447.698,A -85,B 0,C 180,E1 -17353.219,E2 -17353.219} C_VEL
LIN {X 0,Y 278.366,Z 455.72,A -85,B 0,C 180,E1 -17355.376,E2 -17355.376} C_VEL
LIN {X 0,Y 277.095,Z 462.152,A -85,B 0,C 180,E1 -17357.55,E2 -17357.55} C_VEL
LIN {X 0,Y 276.26,Z 467.267,A -85,B 0,C 180,E1 -17359.742,E2 -17359.742} C_VEL
LIN {X 0,Y 275.714,Z 471.242,A -85,B 0,C 180,E1 -17361.94,E2 -17361.94} C_VEL
LIN {X 0,Y 275.322,Z 474.628,A -85,B 0,C 180,E1 -17364.583,E2 -17364.583} C_VEL
LIN {X 0,Y 275.261,Z 476.58,A -85,B 0,C 180,E1 -17367.072,E2 -17367.072} C_VEL
LIN {X 0,Y 275.253,Z 477.19,A -85,B 0,C 180,E1 -17368.536,E2 -17368.536} C_VEL
LIN {X 0,Y 275.251,Z 477.405,A -85,B 0,C 180,E1 -17369.999,E2 -17369.999} C_VEL
LIN {X 0,Y 275.253,Z 477.185,A -85,B 0,C 180,E1 -17371.462,E2 -17371.462} C_VEL
LIN {X 0,Y 275.26,Z 476.572,A -85,B 0,C 180,E1 -17372.926,E2 -17372.926} C_VEL
LIN {X 0,Y 275.328,Z 474.602,A -85,B 0,C 180,E1 -17375.429,E2 -17375.429} C_VEL
LIN {X 0,Y 275.707,Z 471.218,A -85,B 0,C 180,E1 -17378.059,E2 -17378.059} C_VEL
LIN {X 0,Y 276.26,Z 467.232,A -85,B 0,C 180,E1 -17380.257,E2 -17380.257} C_VEL
LIN {X 0,Y 277.272,Z 461.107,A -85,B 0,C 180,E1 -17382.813,E2 -17382.813} C_VEL
LIN {X 0,Y 278.625,Z 454.423,A -85,B 0,C 180,E1 -17384.983,E2 -17384.983} C_VEL
LIN {X 0,Y 280.271,Z 446.134,A -85,B 0,C 180,E1 -17387.135,E2 -17387.135} C_VEL
LIN {X 0,Y 281.733,Z 437.631,A -85,B 0,C 180,E1 -17388.922,E2 -17388.922} C_VEL
LIN {X 0,Y 283.604,Z 427.133,A -85,B 0,C 180,E1 -17390.678,E2 -17390.678} C_VEL
LIN {X 0,Y 285.004,Z 418.224,A -85,B 0,C 180,E1 -17391.891,E2 -17391.891} C_VEL
LIN {X 0,Y 284.273,Z 407.05,A -85,B 0,C 180,E1 -17393.3,E2 -17393.3} C_VEL
LIN {X 0,Y 282.651,Z 394.331,A -85,B 0,C 180,E1 -17394.642,E2 -17394.642} C_VEL
LIN {X 0,Y 279.945,Z 381.076,A -85,B 0,C 180,E1 -17395.793,E2 -17395.793} C_VEL
LIN {X 0,Y 277.285,Z 370.589,A -85,B 0,C 180,E1 -17396.571,E2 -17396.571} C_VEL
LIN {X 0,Y 278.154,Z 365.126,A -85,B 0,C 180,E1 -17400.788,E2 -17400.788} C_VEL
LIN {X 0,Y 278.958,Z 360.376,A -85,B 0,C 180,E1 -17404.529,E2 -17404.529} C_VEL
LIN {X 0,Y 279.098,Z 357.16,A -85,B 0,C 180,E1 -17407.18,E2 -17407.18} C_VEL
LIN {X 0,Y 278.883,Z 353.993,A -85,B 0,C 180,E1 -17409.924,E2 -17409.924} C_VEL
LIN {X 0,Y 278.118,Z 349.645,A -85,B 0,C 180,E1 -17413.963,E2 -17413.963} C_VEL
LIN {X 0,Y 277.271,Z 345.125,A -85,B 0,C 180,E1 -17418.533,E2 -17418.533} C_VEL
LIN {X 0,Y 277.249,Z 344.95,A -85,B 0,C 180,E1 -17422.528,E2 -17422.528} C_VEL
LIN {X 0,Y 277.239,Z 344.952,A -85,B 0,C 180,E1 -17426.103,E2 -17426.103} C_VEL
LIN {X 0,Y 277.255,Z 344.948,A -85,B 0,C 180,E1 -17429.538,E2 -17429.538} C_VEL
LIN {X 0,Y 277.285,Z 344.946,A -85,B 0,C 180,E1 -17432.856,E2 -17432.856} C_VEL
LIN {X 0,Y 277.277,Z 344.948,A -85,B 0,C 180,E1 -17436.075,E2 -17436.075} C_VEL
LIN {X 0,Y 277.337,Z 344.938,A -85,B 0,C 180,E1 -17440.766,E2 -17440.766} C_VEL
LIN {X 0,Y 277.42,Z 344.927,A -85,B 0,C 180,E1 -17445.325,E2 -17445.325} C_VEL
LIN {X 0,Y 277.499,Z 344.919,A -85,B 0,C 180,E1 -17449.788,E2 -17449.788} C_VEL
LIN {X 0,Y 277.646,Z 344.898,A -85,B 0,C 180,E1 -17452.729,E2 -17452.729} C_VEL
LIN {X 0,Y 277.81,Z 344.878,A -85,B 0,C 180,E1 -17458.55,E2 -17458.55} C_VEL
LIN {X 0,Y 277.809,Z 344.881,A -85,B 0,C 180,E1 -17461.45,E2 -17461.45} C_VEL
LIN {X 0,Y 277.646,Z 344.901,A -85,B 0,C 180,E1 -17467.271,E2 -17467.271} C_VEL
LIN {X 0,Y 277.499,Z 344.917,A -85,B 0,C 180,E1 -17470.212,E2 -17470.212} C_VEL
LIN {X 0,Y 277.427,Z 344.925,A -85,B 0,C 180,E1 -17474.675,E2 -17474.675} C_VEL
LIN {X 0,Y 277.338,Z 344.94,A -85,B 0,C 180,E1 -17479.234,E2 -17479.234} C_VEL
LIN {X 0,Y 277.278,Z 344.944,A -85,B 0,C 180,E1 -17483.925,E2 -17483.925} C_VEL
LIN {X 0,Y 277.263,Z 344.947,A -85,B 0,C 180,E1 -17487.483,E2 -17487.483} C_VEL
LIN {X 0,Y 277.242,Z 344.951,A -85,B 0,C 180,E1 -17490.474,E2 -17490.474} C_VEL
LIN {X 0,Y 277.24,Z 344.949,A -85,B 0,C 180,E1 -17493.897,E2 -17493.897} C_VEL
LIN {X 0,Y 277.254,Z 344.947,A -85,B 0,C 180,E1 -17497.472,E2 -17497.472} C_VEL
LIN {X 0,Y 277.179,Z 344.957,A -85,B 0,C 180,E1 -17501.242,E2 -17501.242} C_VEL
LIN {X 0,Y 277.2,Z 344.955,A -85,B 0,C 180,E1 -17505.227,E2 -17505.227} C_VEL
LIN {X 0,Y 277.224,Z 344.954,A -85,B 0,C 180,E1 -17508.768,E2 -17508.768} C_VEL
LIN {X 0,Y 277.252,Z 345.08,A -85,B 0,C 180,E1 -17510.677,E2 -17510.677} C_VEL
LIN {X 0,Y 277.446,Z 347.906,A -85,B 0,C 180,E1 -17514.154,E2 -17514.154} C_VEL
LIN {X 0,Y 277.191,Z 351.135,A -85,B 0,C 180,E1 -17517.831,E2 -17517.831} C_VEL
LIN {X 0,Y 276.9,Z 354.216,A -85,B 0,C 180,E1 -17521.17,E2 -17521.17} C_VEL
LIN {X 0,Y 276.71,Z 356.409,A -85,B 0,C 180,E1 -17523.459,E2 -17523.459} C_VEL
LIN {X 0,Y 281.307,Z 371.204,A -85,B 0,C 180,E1 -17524.724,E2 -17524.724} C_VEL
LIN {X 0,Y 284.286,Z 383.498,A -85,B 0,C 180,E1 -17525.973,E2 -17525.973} C_VEL
LIN {X 0,Y 286.118,Z 394.181,A -85,B 0,C 180,E1 -17527.241,E2 -17527.241} C_VEL
LIN {X 0,Y 286.392,Z 398.875,A -85,B 0,C 180,E1 -17527.835,E2 -17527.835} C_VEL
LIN {X 0,Y 284.725,Z 409.531,A -85,B 0,C 180,E1 -17529.218,E2 -17529.218} C_VEL
LIN {X 0,Y 283.134,Z 419.93,A -85,B 0,C 180,E1 -17530.935,E2 -17530.935} C_VEL
LIN {X 0,Y 281.228,Z 429.656,A -85,B 0,C 180,E1 -17532.925,E2 -17532.925} C_VEL
LIN {X 0,Y 279.504,Z 437.901,A -85,B 0,C 180,E1 -17535.065,E2 -17535.065} C_VEL
LIN {X 0,Y 278.362,Z 443.538,A -85,B 0,C 180,E1 -17536.867,E2 -17536.867} C_VEL
LIN {X 0,Y 277.239,Z 449.032,A -85,B 0,C 180,E1 -17539.041,E2 -17539.041} C_VEL
LIN {X 0,Y 276.403,Z 453.342,A -85,B 0,C 180,E1 -17541.226,E2 -17541.226} C_VEL
LIN {X 0,Y 275.945,Z 456.516,A -85,B 0,C 180,E1 -17543.359,E2 -17543.359} C_VEL
LIN {X 0,Y 275.579,Z 458.865,A -85,B 0,C 180,E1 -17545.613,E2 -17545.613} C_VEL
LIN {X 0,Y 275.431,Z 459.856,A -85,B 0,C 180,E1 -17547.075,E2 -17547.075} C_VEL
LIN {X 0,Y 275.288,Z 460.696,A -85,B 0,C 180,E1 -17550.001,E2 -17550.001} C_VEL
LIN {X 0,Y 275.315,Z 460.503,A -85,B 0,C 180,E1 -17551.463,E2 -17551.463} C_VEL
LIN {X 0,Y 275.428,Z 459.916,A -85,B 0,C 180,E1 -17552.926,E2 -17552.926} C_VEL
LIN {X 0,Y 275.767,Z 457.592,A -85,B 0,C 180,E1 -17555.851,E2 -17555.851} C_VEL
LIN {X 0,Y 276.239,Z 454.726,A -85,B 0,C 180,E1 -17558.044,E2 -17558.044} C_VEL
LIN {X 0,Y 276.874,Z 450.841,A -85,B 0,C 180,E1 -17560.235,E2 -17560.235} C_VEL
LIN {X 0,Y 277.896,Z 445.823,A -85,B 0,C 180,E1 -17562.414,E2 -17562.414} C_VEL
LIN {X 0,Y 279.161,Z 439.504,A -85,B 0,C 180,E1 -17564.582,E2 -17564.582} C_VEL
LIN {X 0,Y 280.892,Z 431.59,A -85,B 0,C 180,E1 -17566.723,E2 -17566.723} C_VEL
LIN {X 0,Y 282.78,Z 421.749,A -85,B 0,C 180,E1 -17568.85,E2 -17568.85} C_VEL
LIN {X 0,Y 284.26,Z 412.587,A -85,B 0,C 180,E1 -17570.44,E2 -17570.44} C_VEL
LIN {X 0,Y 286.104,Z 401.177,A -85,B 0,C 180,E1 -17572,E2 -17572} C_VEL
LIN {X 0,Y 286.471,Z 398.272,A -85,B 0,C 180,E1 -17572.35,E2 -17572.35} C_VEL
LIN {X 0,Y 285.136,Z 388.038,A -85,B 0,C 180,E1 -17573.628,E2 -17573.628} C_VEL
LIN {X 0,Y 283.136,Z 378.216,A -85,B 0,C 180,E1 -17574.709,E2 -17574.709} C_VEL
LIN {X 0,Y 279.883,Z 366.458,A -85,B 0,C 180,E1 -17575.835,E2 -17575.835} C_VEL
LIN {X 0,Y 276.722,Z 356.412,A -85,B 0,C 180,E1 -17576.662,E2 -17576.662} C_VEL
LIN {X 0,Y 277.045,Z 352.781,A -85,B 0,C 180,E1 -17580.488,E2 -17580.488} C_VEL
LIN {X 0,Y 277.338,Z 349.744,A -85,B 0,C 180,E1 -17583.883,E2 -17583.883} C_VEL
LIN {X 0,Y 277.454,Z 348.052,A -85,B 0,C 180,E1 -17585.848,E2 -17585.848} C_VEL
LIN {X 0,Y 277.256,Z 345.189,A -85,B 0,C 180,E1 -17589.324,E2 -17589.324} C_VEL
LIN {X 0,Y 277.216,Z 344.956,A -85,B 0,C 180,E1 -17592.675,E2 -17592.675} C_VEL
LIN {X 0,Y 277.19,Z 344.958,A -85,B 0,C 180,E1 -17596.798,E2 -17596.798} C_VEL
LIN {X 0,Y 277.196,Z 344.955,A -85,B 0,C 180,E1 -17600.665,E2 -17600.665} C_VEL
LIN {X 0,Y 277.281,Z 344.944,A -85,B 0,C 180,E1 -17604.341,E2 -17604.341} C_VEL
LIN {X 0,Y 277.239,Z 344.948,A -85,B 0,C 180,E1 -17607.835,E2 -17607.835} C_VEL
LIN {X 0,Y 277.238,Z 344.95,A -85,B 0,C 180,E1 -17611.206,E2 -17611.206} C_VEL
LIN {X 0,Y 277.245,Z 344.948,A -85,B 0,C 180,E1 -17614.473,E2 -17614.473} C_VEL
LIN {X 0,Y 277.265,Z 344.946,A -85,B 0,C 180,E1 -17617.653,E2 -17617.653} C_VEL
LIN {X 0,Y 277.343,Z 344.939,A -85,B 0,C 180,E1 -17620.766,E2 -17620.766} C_VEL
LIN {X 0,Y 277.433,Z 344.925,A -85,B 0,C 180,E1 -17625.326,E2 -17625.326} C_VEL
LIN {X 0,Y 277.505,Z 344.916,A -85,B 0,C 180,E1 -17629.789,E2 -17629.789} C_VEL
LIN {X 0,Y 277.652,Z 344.9,A -85,B 0,C 180,E1 -17632.729,E2 -17632.729} C_VEL
LIN {X 0,Y 277.814,Z 344.88,A -85,B 0,C 180,E1 -17638.55,E2 -17638.55} C_VEL
LIN {X 0,Y 277.814,Z 344.877,A -85,B 0,C 180,E1 -17641.45,E2 -17641.45} C_VEL
LIN {X 0,Y 277.639,Z 344.9,A -85,B 0,C 180,E1 -17647.271,E2 -17647.271} C_VEL
LIN {X 0,Y 277.499,Z 344.917,A -85,B 0,C 180,E1 -17649.655,E2 -17649.655} C_VEL
LIN {X 0,Y 276.763,Z 345.013,A -85,B 0,C 180,E1 -17650.865,E2 -17650.865} C_VEL
LIN {X 0,Y 273.901,Z 345.375,A -85,B 0,C 180,E1 -17652.838,E2 -17652.838} C_VEL
LIN {X 0,Y 271.503,Z 345.672,A -85,B 0,C 180,E1 -17654.44,E2 -17654.44} C_VEL
LIN {X 0,Y 270.459,Z 345.799,A -85,B 0,C 180,E1 -17655.681,E2 -17655.681} C_VEL
LIN {X 0,Y 270.363,Z 345.809,A -85,B 0,C 180,E1 -17656.102,E2 -17656.102} C_VEL
LIN {X 0,Y 270.29,Z 345.816,A -85,B 0,C 180,E1 -17660.601,E2 -17660.601} C_VEL
LIN {X 0,Y 270.223,Z 345.823,A -85,B 0,C 180,E1 -17664.591,E2 -17664.591} C_VEL
LIN {X 0,Y 270.197,Z 345.83,A -85,B 0,C 180,E1 -17667.917,E2 -17667.917} C_VEL
LIN {X 0,Y 270.172,Z 345.834,A -85,B 0,C 180,E1 -17671.35,E2 -17671.35} C_VEL
LIN {X 0,Y 270.197,Z 345.831,A -85,B 0,C 180,E1 -17674.906,E2 -17674.906} C_VEL
LIN {X 0,Y 270.197,Z 345.829,A -85,B 0,C 180,E1 -17678.711,E2 -17678.711} C_VEL
LIN {X 0,Y 270.198,Z 346.051,A -85,B 0,C 180,E1 -17680.903,E2 -17680.903} C_VEL
LIN {X 0,Y 270.786,Z 349.438,A -85,B 0,C 180,E1 -17684.488,E2 -17684.488} C_VEL
LIN {X 0,Y 271.579,Z 353.667,A -85,B 0,C 180,E1 -17688.631,E2 -17688.631} C_VEL
LIN {X 0,Y 271.949,Z 356.981,A -85,B 0,C 180,E1 -17691.667,E2 -17691.667} C_VEL
LIN {X 0,Y 271.969,Z 360.181,A -85,B 0,C 180,E1 -17694.449,E2 -17694.449} C_VEL
LIN {X 0,Y 271.575,Z 363.374,A -85,B 0,C 180,E1 -17697.081,E2 -17697.081} C_VEL
LIN {X 0,Y 270.648,Z 368.618,A -85,B 0,C 180,E1 -17701.29,E2 -17701.29} C_VEL
LIN {X 0,Y 270.365,Z 370.392,A -85,B 0,C 180,E1 -17702.697,E2 -17702.697} C_VEL
LIN {X 0,Y 272.432,Z 378.442,A -85,B 0,C 180,E1 -17703.281,E2 -17703.281} C_VEL
LIN {X 0,Y 275.214,Z 390.802,A -85,B 0,C 180,E1 -17704.364,E2 -17704.364} C_VEL
LIN {X 0,Y 276.944,Z 401.964,A -85,B 0,C 180,E1 -17705.511,E2 -17705.511} C_VEL
LIN {X 0,Y 277.94,Z 412.865,A -85,B 0,C 180,E1 -17706.824,E2 -17706.824} C_VEL
LIN {X 0,Y 278.113,Z 420.841,A -85,B 0,C 180,E1 -17707.92,E2 -17707.92} C_VEL
LIN {X 0,Y 276.146,Z 431.492,A -85,B 0,C 180,E1 -17709.516,E2 -17709.516} C_VEL
LIN {X 0,Y 274.445,Z 440.711,A -85,B 0,C 180,E1 -17711.247,E2 -17711.247} C_VEL
LIN {X 0,Y 272.809,Z 448.972,A -85,B 0,C 180,E1 -17713.153,E2 -17713.153} C_VEL
LIN {X 0,Y 271.223,Z 456.664,A -85,B 0,C 180,E1 -17715.366,E2 -17715.366} C_VEL
LIN {X 0,Y 269.82,Z 463.762,A -85,B 0,C 180,E1 -17717.972,E2 -17717.972} C_VEL
LIN {X 0,Y 269.015,Z 468.487,A -85,B 0,C 180,E1 -17720.223,E2 -17720.223} C_VEL
LIN {X 0,Y 268.5,Z 472.1,A -85,B 0,C 180,E1 -17722.479,E2 -17722.479} C_VEL
LIN {X 0,Y 268.213,Z 474.663,A -85,B 0,C 180,E1 -17724.697,E2 -17724.697} C_VEL
LIN {X 0,Y 268.174,Z 476.365,A -85,B 0,C 180,E1 -17726.995,E2 -17726.995} C_VEL
LIN {X 0,Y 268.18,Z 476.975,A -85,B 0,C 180,E1 -17728.498,E2 -17728.498} C_VEL
LIN {X 0,Y 268.176,Z 477.19,A -85,B 0,C 180,E1 -17729.999,E2 -17729.999} C_VEL
LIN {X 0,Y 268.179,Z 476.97,A -85,B 0,C 180,E1 -17731.501,E2 -17731.501} C_VEL
LIN {X 0,Y 268.173,Z 476.357,A -85,B 0,C 180,E1 -17733.004,E2 -17733.004} C_VEL
LIN {X 0,Y 268.226,Z 474.618,A -85,B 0,C 180,E1 -17735.333,E2 -17735.333} C_VEL
LIN {X 0,Y 268.64,Z 471.001,A -85,B 0,C 180,E1 -17738.272,E2 -17738.272} C_VEL
LIN {X 0,Y 269.258,Z 467.015,A -85,B 0,C 180,E1 -17740.527,E2 -17740.527} C_VEL
LIN {X 0,Y 270.326,Z 460.889,A -85,B 0,C 180,E1 -17743.148,E2 -17743.148} C_VEL
LIN {X 0,Y 271.761,Z 454.206,A -85,B 0,C 180,E1 -17745.37,E2 -17745.37} C_VEL
LIN {X 0,Y 273.482,Z 445.915,A -85,B 0,C 180,E1 -17747.574,E2 -17747.574} C_VEL
LIN {X 0,Y 274.988,Z 437.411,A -85,B 0,C 180,E1 -17749.404,E2 -17749.404} C_VEL
LIN {X 0,Y 276.965,Z 426.913,A -85,B 0,C 180,E1 -17751.197,E2 -17751.197} C_VEL
LIN {X 0,Y 278.247,Z 419.381,A -85,B 0,C 180,E1 -17752.263,E2 -17752.263} C_VEL
LIN {X 0,Y 277.603,Z 408.373,A -85,B 0,C 180,E1 -17753.722,E2 -17753.722} C_VEL
LIN {X 0,Y 276.143,Z 396.142,A -85,B 0,C 180,E1 -17755.083,E2 -17755.083} C_VEL
LIN {X 0,Y 273.7,Z 383.54,A -85,B 0,C 180,E1 -17756.27,E2 -17756.27} C_VEL
LIN {X 0,Y 270.364,Z 370.377,A -85,B 0,C 180,E1 -17757.29,E2 -17757.29} C_VEL
LIN {X 0,Y 271.174,Z 365.454,A -85,B 0,C 180,E1 -17761.219,E2 -17761.219} C_VEL
LIN {X 0,Y 271.938,Z 361.225,A -85,B 0,C 180,E1 -17764.649,E2 -17764.649} C_VEL
LIN {X 0,Y 272.045,Z 358.7,A -85,B 0,C 180,E1 -17766.788,E2 -17766.788} C_VEL
LIN {X 0,Y 271.833,Z 354.799,A -85,B 0,C 180,E1 -17770.265,E2 -17770.265} C_VEL
LIN {X 0,Y 271.04,Z 350.481,A -85,B 0,C 180,E1 -17774.433,E2 -17774.433} C_VEL
LIN {X 0,Y 270.5,Z 347.481,A -85,B 0,C 180,E1 -17777.505,E2 -17777.505} C_VEL
LIN {X 0,Y 270.166,Z 345.836,A -85,B 0,C 180,E1 -17779.433,E2 -17779.433} C_VEL
LIN {X 0,Y 270.203,Z 345.828,A -85,B 0,C 180,E1 -17783.257,E2 -17783.257} C_VEL
LIN {X 0,Y 270.195,Z 345.831,A -85,B 0,C 180,E1 -17786.891,E2 -17786.891} C_VEL
LIN {X 0,Y 270.176,Z 345.834,A -85,B 0,C 180,E1 -17790.38,E2 -17790.38} C_VEL
LIN {X 0,Y 270.196,Z 345.829,A -85,B 0,C 180,E1 -17793.757,E2 -17793.757} C_VEL
LIN {X 0,Y 270.197,Z 345.827,A -85,B 0,C 180,E1 -17797.036,E2 -17797.036} C_VEL
LIN {X 0,Y 270.294,Z 345.817,A -85,B 0,C 180,E1 -17800.244,E2 -17800.244} C_VEL
LIN {X 0,Y 270.389,Z 345.803,A -85,B 0,C 180,E1 -17804.935,E2 -17804.935} C_VEL
LIN {X 0,Y 270.434,Z 345.797,A -85,B 0,C 180,E1 -17809.519,E2 -17809.519} C_VEL
LIN {X 0,Y 270.604,Z 345.776,A -85,B 0,C 180,E1 -17812.539,E2 -17812.539} C_VEL
LIN {X 0,Y 270.776,Z 345.754,A -85,B 0,C 180,E1 -17818.513,E2 -17818.513} C_VEL
LIN {X 0,Y 270.775,Z 345.758,A -85,B 0,C 180,E1 -17821.487,E2 -17821.487} C_VEL
LIN {X 0,Y 270.604,Z 345.779,A -85,B 0,C 180,E1 -17827.461,E2 -17827.461} C_VEL
LIN {X 0,Y 270.434,Z 345.797,A -85,B 0,C 180,E1 -17830.481,E2 -17830.481} C_VEL
LIN {X 0,Y 270.396,Z 345.803,A -85,B 0,C 180,E1 -17835.065,E2 -17835.065} C_VEL
LIN {X 0,Y 270.295,Z 345.815,A -85,B 0,C 180,E1 -17839.756,E2 -17839.756} C_VEL
LIN {X 0,Y 270.218,Z 345.825,A -85,B 0,C 180,E1 -17844.591,E2 -17844.591} C_VEL
LIN {X 0,Y 270.192,Z 345.827,A -85,B 0,C 180,E1 -17847.918,E2 -17847.918} C_VEL
LIN {X 0,Y 270.167,Z 345.832,A -85,B 0,C 180,E1 -17851.351,E2 -17851.351} C_VEL
LIN {X 0,Y 270.193,Z 345.831,A -85,B 0,C 180,E1 -17854.907,E2 -17854.907} C_VEL
LIN {X 0,Y 270.193,Z 345.83,A -85,B 0,C 180,E1 -17858.712,E2 -17858.712} C_VEL
LIN {X 0,Y 270.144,Z 345.833,A -85,B 0,C 180,E1 -17863.246,E2 -17863.246} C_VEL
LIN {X 0,Y 270.187,Z 345.83,A -85,B 0,C 180,E1 -17867.447,E2 -17867.447} C_VEL
LIN {X 0,Y 270.181,Z 345.831,A -85,B 0,C 180,E1 -17869.437,E2 -17869.437} C_VEL
LIN {X 0,Y 270.312,Z 346.798,A -85,B 0,C 180,E1 -17871.394,E2 -17871.394} C_VEL
LIN {X 0,Y 270.419,Z 348.618,A -85,B 0,C 180,E1 -17873.675,E2 -17873.675} C_VEL
LIN {X 0,Y 270.25,Z 351.343,A -85,B 0,C 180,E1 -17876.901,E2 -17876.901} C_VEL
LIN {X 0,Y 269.935,Z 354.44,A -85,B 0,C 180,E1 -17880.353,E2 -17880.353} C_VEL
LIN {X 0,Y 269.722,Z 356.622,A -85,B 0,C 180,E1 -17882.716,E2 -17882.716} C_VEL
LIN {X 0,Y 274.298,Z 370.941,A -85,B 0,C 180,E1 -17883.996,E2 -17883.996} C_VEL
LIN {X 0,Y 277.292,Z 382.901,A -85,B 0,C 180,E1 -17885.252,E2 -17885.252} C_VEL
LIN {X 0,Y 279.283,Z 394.456,A -85,B 0,C 180,E1 -17886.657,E2 -17886.657} C_VEL
LIN {X 0,Y 279.741,Z 399.119,A -85,B 0,C 180,E1 -17887.281,E2 -17887.281} C_VEL
LIN {X 0,Y 278.111,Z 409.75,A -85,B 0,C 180,E1 -17888.7,E2 -17888.7} C_VEL
LIN {X 0,Y 276.544,Z 419.389,A -85,B 0,C 180,E1 -17890.311,E2 -17890.311} C_VEL
LIN {X 0,Y 274.806,Z 428.28,A -85,B 0,C 180,E1 -17892.129,E2 -17892.129} C_VEL
LIN {X 0,Y 272.917,Z 436.893,A -85,B 0,C 180,E1 -17894.314,E2 -17894.314} C_VEL
LIN {X 0,Y 271.459,Z 443.755,A -85,B 0,C 180,E1 -17896.527,E2 -17896.527} C_VEL
LIN {X 0,Y 270.261,Z 449.249,A -85,B 0,C 180,E1 -17898.754,E2 -17898.754} C_VEL
LIN {X 0,Y 269.374,Z 453.559,A -85,B 0,C 180,E1 -17900.995,E2 -17900.995} C_VEL
LIN {X 0,Y 268.849,Z 456.983,A -85,B 0,C 180,E1 -17903.397,E2 -17903.397} C_VEL
LIN {X 0,Y 268.508,Z 459.08,A -85,B 0,C 180,E1 -17905.497,E2 -17905.497} C_VEL
LIN {X 0,Y 268.367,Z 460.071,A -85,B 0,C 180,E1 -17906.998,E2 -17906.998} C_VEL
LIN {X 0,Y 268.212,Z 460.91,A -85,B 0,C 180,E1 -17910.001,E2 -17910.001} C_VEL
LIN {X 0,Y 268.243,Z 460.717,A -85,B 0,C 180,E1 -17911.502,E2 -17911.502} C_VEL
LIN {X 0,Y 268.364,Z 460.13,A -85,B 0,C 180,E1 -17913.003,E2 -17913.003} C_VEL
LIN {X 0,Y 268.718,Z 457.807,A -85,B 0,C 180,E1 -17916.006,E2 -17916.006} C_VEL
LIN {X 0,Y 269.201,Z 454.941,A -85,B 0,C 180,E1 -17918.256,E2 -17918.256} C_VEL
LIN {X 0,Y 269.875,Z 451.056,A -85,B 0,C 180,E1 -17920.504,E2 -17920.504} C_VEL
LIN {X 0,Y 270.973,Z 446.037,A -85,B 0,C 180,E1 -17922.736,E2 -17922.736} C_VEL
LIN {X 0,Y 272.284,Z 439.718,A -85,B 0,C 180,E1 -17924.958,E2 -17924.958} C_VEL
LIN {X 0,Y 274.104,Z 431.803,A -85,B 0,C 180,E1 -17927.149,E2 -17927.149} C_VEL
LIN {X 0,Y 275.757,Z 423.736,A -85,B 0,C 180,E1 -17928.963,E2 -17928.963} C_VEL
LIN {X 0,Y 277.45,Z 413.896,A -85,B 0,C 180,E1 -17930.771,E2 -17930.771} C_VEL
LIN {X 0,Y 279.326,Z 402.809,A -85,B 0,C 180,E1 -17932.368,E2 -17932.368} C_VEL
LIN {X 0,Y 279.733,Z 398.488,A -85,B 0,C 180,E1 -17932.919,E2 -17932.919} C_VEL
LIN {X 0,Y 278.195,Z 387.311,A -85,B 0,C 180,E1 -17934.351,E2 -17934.351} C_VEL
LIN {X 0,Y 275.479,Z 375.16,A -85,B 0,C 180,E1 -17935.703,E2 -17935.703} C_VEL
LIN {X 0,Y 271.637,Z 362.481,A -85,B 0,C 180,E1 -17936.918,E2 -17936.918} C_VEL
LIN {X 0,Y 269.689,Z 356.64,A -85,B 0,C 180,E1 -17937.397,E2 -17937.397} C_VEL
LIN {X 0,Y 270.085,Z 353,A -85,B 0,C 180,E1 -17941.361,E2 -17941.361} C_VEL
LIN {X 0,Y 270.36,Z 349.971,A -85,B 0,C 180,E1 -17944.882,E2 -17944.882} C_VEL
LIN {X 0,Y 270.414,Z 348.437,A -85,B 0,C 180,E1 -17946.71,E2 -17946.71} C_VEL
LIN {X 0,Y 270.31,Z 346.809,A -85,B 0,C 180,E1 -17948.74,E2 -17948.74} C_VEL
LIN {X 0,Y 270.17,Z 345.834,A -85,B 0,C 180,E1 -17951.028,E2 -17951.028} C_VEL
LIN {X 0,Y 270.15,Z 345.836,A -85,B 0,C 180,E1 -17954.62,E2 -17954.62} C_VEL
LIN {X 0,Y 270.15,Z 345.836,A -85,B 0,C 180,E1 -17957.437,E2 -17957.437} C_VEL
LIN {X 0,Y 270.167,Z 345.833,A -85,B 0,C 180,E1 -17961.367,E2 -17961.367} C_VEL
LIN {X 0,Y 270.2,Z 345.828,A -85,B 0,C 180,E1 -17965.094,E2 -17965.094} C_VEL
LIN {X 0,Y 270.183,Z 345.831,A -85,B 0,C 180,E1 -17969.136,E2 -17969.136} C_VEL
LIN {X 0,Y 270.221,Z 345.823,A -85,B 0,C 180,E1 -17972.163,E2 -17972.163} C_VEL
LIN {X 0,Y 270.226,Z 345.823,A -85,B 0,C 180,E1 -17975.542,E2 -17975.542} C_VEL
LIN {X 0,Y 270.3,Z 345.814,A -85,B 0,C 180,E1 -17980.244,E2 -17980.244} C_VEL
LIN {X 0,Y 270.402,Z 345.803,A -85,B 0,C 180,E1 -17984.935,E2 -17984.935} C_VEL
LIN {X 0,Y 270.44,Z 345.796,A -85,B 0,C 180,E1 -17989.519,E2 -17989.519} C_VEL
LIN {X 0,Y 270.61,Z 345.778,A -85,B 0,C 180,E1 -17992.539,E2 -17992.539} C_VEL
LIN {X 0,Y 270.781,Z 345.756,A -85,B 0,C 180,E1 -17998.513,E2 -17998.513} C_VEL
LIN {X 0,Y 270.78,Z 345.753,A -85,B 0,C 180,E1 -18001.487,E2 -18001.487} C_VEL
LIN {X 0,Y 270.597,Z 345.778,A -85,B 0,C 180,E1 -18007.462,E2 -18007.462} C_VEL
LIN {X 0,Y 270.411,Z 345.802,A -85,B 0,C 180,E1 -18010.482,E2 -18010.482} C_VEL
LIN {X 0,Y 270.395,Z 345.803,A -85,B 0,C 180,E1 -18015.065,E2 -18015.065} C_VEL
LIN {X 0,Y 270.363,Z 345.809,A -85,B 0,C 180,E1 -18016.102,E2 -18016.102} C_VEL
LIN {X 0,Y 269.647,Z 345.898,A -85,B 0,C 180,E1 -18017.346,E2 -18017.346} C_VEL
LIN {X 0,Y 266.717,Z 346.263,A -85,B 0,C 180,E1 -18019.371,E2 -18019.371} C_VEL
LIN {X 0,Y 264.252,Z 346.568,A -85,B 0,C 180,E1 -18021.017,E2 -18021.017} C_VEL
LIN {X 0,Y 263.2,Z 346.699,A -85,B 0,C 180,E1 -18022.296,E2 -18022.296} C_VEL
LIN {X 0,Y 263.117,Z 346.708,A -85,B 0,C 180,E1 -18022.729,E2 -18022.729} C_VEL
LIN {X 0,Y 263.166,Z 346.705,A -85,B 0,C 180,E1 -18025.296,E2 -18025.296} C_VEL
LIN {X 0,Y 263.132,Z 346.708,A -85,B 0,C 180,E1 -18028.735,E2 -18028.735} C_VEL
LIN {X 0,Y 263.127,Z 346.71,A -85,B 0,C 180,E1 -18032.289,E2 -18032.289} C_VEL
LIN {X 0,Y 263.175,Z 346.704,A -85,B 0,C 180,E1 -18036.761,E2 -18036.761} C_VEL
LIN {X 0,Y 263.127,Z 346.756,A -85,B 0,C 180,E1 -18040.118,E2 -18040.118} C_VEL
LIN {X 0,Y 263.734,Z 350.298,A -85,B 0,C 180,E1 -18043.987,E2 -18043.987} C_VEL
LIN {X 0,Y 264.541,Z 354.616,A -85,B 0,C 180,E1 -18048.381,E2 -18048.381} C_VEL
LIN {X 0,Y 264.928,Z 357.835,A -85,B 0,C 180,E1 -18051.435,E2 -18051.435} C_VEL
LIN {X 0,Y 264.884,Z 362.238,A -85,B 0,C 180,E1 -18055.336,E2 -18055.336} C_VEL
LIN {X 0,Y 263.938,Z 367.35,A -85,B 0,C 180,E1 -18059.607,E2 -18059.607} C_VEL
LIN {X 0,Y 263.472,Z 370.173,A -85,B 0,C 180,E1 -18061.921,E2 -18061.921} C_VEL
LIN {X 0,Y 265.727,Z 378.841,A -85,B 0,C 180,E1 -18062.587,E2 -18062.587} C_VEL
LIN {X 0,Y 268.487,Z 390.99,A -85,B 0,C 180,E1 -18063.705,E2 -18063.705} C_VEL
LIN {X 0,Y 270.228,Z 402.103,A -85,B 0,C 180,E1 -18064.898,E2 -18064.898} C_VEL
LIN {X 0,Y 271.21,Z 413.258,A -85,B 0,C 180,E1 -18066.292,E2 -18066.292} C_VEL
LIN {X 0,Y 271.299,Z 421.923,A -85,B 0,C 180,E1 -18067.536,E2 -18067.536} C_VEL
LIN {X 0,Y 269.289,Z 432.352,A -85,B 0,C 180,E1 -18069.17,E2 -18069.17} C_VEL
LIN {X 0,Y 267.398,Z 442.151,A -85,B 0,C 180,E1 -18071.118,E2 -18071.118} C_VEL
LIN {X 0,Y 265.675,Z 450.135,A -85,B 0,C 180,E1 -18073.083,E2 -18073.083} C_VEL
LIN {X 0,Y 264.104,Z 457.572,A -85,B 0,C 180,E1 -18075.356,E2 -18075.356} C_VEL
LIN {X 0,Y 262.827,Z 463.546,A -85,B 0,C 180,E1 -18077.647,E2 -18077.647} C_VEL
LIN {X 0,Y 262.007,Z 468.272,A -85,B 0,C 180,E1 -18079.958,E2 -18079.958} C_VEL
LIN {X 0,Y 261.431,Z 471.885,A -85,B 0,C 180,E1 -18082.275,E2 -18082.275} C_VEL
LIN {X 0,Y 261.124,Z 474.654,A -85,B 0,C 180,E1 -18084.769,E2 -18084.769} C_VEL
LIN {X 0,Y 261.089,Z 476.15,A -85,B 0,C 180,E1 -18086.913,E2 -18086.913} C_VEL
LIN {X 0,Y 261.108,Z 476.761,A -85,B 0,C 180,E1 -18088.457,E2 -18088.457} C_VEL
LIN {X 0,Y 261.103,Z 476.975,A -85,B 0,C 180,E1 -18089.999,E2 -18089.999} C_VEL
LIN {X 0,Y 261.107,Z 476.755,A -85,B 0,C 180,E1 -18091.542,E2 -18091.542} C_VEL
LIN {X 0,Y 261.089,Z 476.141,A -85,B 0,C 180,E1 -18093.085,E2 -18093.085} C_VEL
LIN {X 0,Y 261.23,Z 473.732,A -85,B 0,C 180,E1 -18096.177,E2 -18096.177} C_VEL
LIN {X 0,Y 261.588,Z 470.783,A -85,B 0,C 180,E1 -18098.497,E2 -18098.497} C_VEL
LIN {X 0,Y 262.252,Z 466.797,A -85,B 0,C 180,E1 -18100.811,E2 -18100.811} C_VEL
LIN {X 0,Y 263.394,Z 460.671,A -85,B 0,C 180,E1 -18103.501,E2 -18103.501} C_VEL
LIN {X 0,Y 264.908,Z 453.988,A -85,B 0,C 180,E1 -18105.778,E2 -18105.778} C_VEL
LIN {X 0,Y 266.7,Z 445.697,A -85,B 0,C 180,E1 -18108.036,E2 -18108.036} C_VEL
LIN {X 0,Y 268.263,Z 437.191,A -85,B 0,C 180,E1 -18109.911,E2 -18109.911} C_VEL
LIN {X 0,Y 270.36,Z 426.694,A -85,B 0,C 180,E1 -18111.741,E2 -18111.741} C_VEL
LIN {X 0,Y 271.47,Z 420.481,A -85,B 0,C 180,E1 -18112.648,E2 -18112.648} C_VEL
LIN {X 0,Y 270.903,Z 409.227,A -85,B 0,C 180,E1 -18114.221,E2 -18114.221} C_VEL
LIN {X 0,Y 269.591,Z 397.664,A -85,B 0,C 180,E1 -18115.578,E2 -18115.578} C_VEL
LIN {X 0,Y 267.212,Z 384.813,A -85,B 0,C 180,E1 -18116.855,E2 -18116.855} C_VEL
LIN {X 0,Y 263.708,Z 371.702,A -85,B 0,C 180,E1 -18117.963,E2 -18117.963} C_VEL
LIN {X 0,Y 263.473,Z 370.098,A -85,B 0,C 180,E1 -18118.113,E2 -18118.113} C_VEL
LIN {X 0,Y 264.306,Z 365.237,A -85,B 0,C 180,E1 -18122.126,E2 -18122.126} C_VEL
LIN {X 0,Y 264.883,Z 362.2,A -85,B 0,C 180,E1 -18124.663,E2 -18124.663} C_VEL
LIN {X 0,Y 265.001,Z 358.876,A -85,B 0,C 180,E1 -18127.586,E2 -18127.586} C_VEL
LIN {X 0,Y 264.895,Z 356.564,A -85,B 0,C 180,E1 -18129.699,E2 -18129.699} C_VEL
LIN {X 0,Y 264.194,Z 352.419,A -85,B 0,C 180,E1 -18133.758,E2 -18133.758} C_VEL
LIN {X 0,Y 263.388,Z 348.096,A -85,B 0,C 180,E1 -18138.34,E2 -18138.34} C_VEL
LIN {X 0,Y 263.099,Z 346.714,A -85,B 0,C 180,E1 -18140.126,E2 -18140.126} C_VEL
LIN {X 0,Y 263.152,Z 346.707,A -85,B 0,C 180,E1 -18144.016,E2 -18144.016} C_VEL
LIN {X 0,Y 263.122,Z 346.71,A -85,B 0,C 180,E1 -18147.71,E2 -18147.71} C_VEL
LIN {X 0,Y 263.141,Z 346.708,A -85,B 0,C 180,E1 -18151.804,E2 -18151.804} C_VEL
LIN {X 0,Y 263.183,Z 346.702,A -85,B 0,C 180,E1 -18155.217,E2 -18155.217} C_VEL
LIN {X 0,Y 263.256,Z 346.692,A -85,B 0,C 180,E1 -18159.693,E2 -18159.693} C_VEL
LIN {X 0,Y 263.337,Z 346.683,A -85,B 0,C 180,E1 -18164.521,E2 -18164.521} C_VEL
LIN {X 0,Y 263.366,Z 346.677,A -85,B 0,C 180,E1 -18169.234,E2 -18169.234} C_VEL
LIN {X 0,Y 263.566,Z 346.654,A -85,B 0,C 180,E1 -18172.338,E2 -18172.338} C_VEL
LIN {X 0,Y 263.741,Z 346.631,A -85,B 0,C 180,E1 -18178.473,E2 -18178.473} C_VEL
LIN {X 0,Y 263.74,Z 346.634,A -85,B 0,C 180,E1 -18181.527,E2 -18181.527} C_VEL
LIN {X 0,Y 263.566,Z 346.654,A -85,B 0,C 180,E1 -18187.662,E2 -18187.662} C_VEL
LIN {X 0,Y 263.366,Z 346.678,A -85,B 0,C 180,E1 -18190.766,E2 -18190.766} C_VEL
LIN {X 0,Y 263.344,Z 346.683,A -85,B 0,C 180,E1 -18195.479,E2 -18195.479} C_VEL
LIN {X 0,Y 263.257,Z 346.691,A -85,B 0,C 180,E1 -18200.307,E2 -18200.307} C_VEL
LIN {X 0,Y 263.161,Z 346.705,A -85,B 0,C 180,E1 -18205.296,E2 -18205.296} C_VEL
LIN {X 0,Y 263.127,Z 346.71,A -85,B 0,C 180,E1 -18208.736,E2 -18208.736} C_VEL
LIN {X 0,Y 263.122,Z 346.709,A -85,B 0,C 180,E1 -18212.29,E2 -18212.29} C_VEL
LIN {X 0,Y 263.173,Z 346.705,A -85,B 0,C 180,E1 -18216.763,E2 -18216.763} C_VEL
LIN {X 0,Y 263.086,Z 346.713,A -85,B 0,C 180,E1 -18219.876,E2 -18219.876} C_VEL
LIN {X 0,Y 263.094,Z 346.712,A -85,B 0,C 180,E1 -18223.99,E2 -18223.99} C_VEL
LIN {X 0,Y 263.139,Z 346.709,A -85,B 0,C 180,E1 -18228.111,E2 -18228.111} C_VEL
LIN {X 0,Y 263.149,Z 347.017,A -85,B 0,C 180,E1 -18230.137,E2 -18230.137} C_VEL
LIN {X 0,Y 263.383,Z 349.342,A -85,B 0,C 180,E1 -18233.179,E2 -18233.179} C_VEL
LIN {X 0,Y 263.296,Z 351.569,A -85,B 0,C 180,E1 -18235.908,E2 -18235.908} C_VEL
LIN {X 0,Y 262.973,Z 354.663,A -85,B 0,C 180,E1 -18239.485,E2 -18239.485} C_VEL
LIN {X 0,Y 262.768,Z 356.835,A -85,B 0,C 180,E1 -18241.905,E2 -18241.905} C_VEL
LIN {X 0,Y 264.586,Z 362.44,A -85,B 0,C 180,E1 -18242.417,E2 -18242.417} C_VEL
LIN {X 0,Y 268.177,Z 373.856,A -85,B 0,C 180,E1 -18243.545,E2 -18243.545} C_VEL
LIN {X 0,Y 270.95,Z 385.519,A -85,B 0,C 180,E1 -18244.867,E2 -18244.867} C_VEL
LIN {X 0,Y 272.764,Z 396.738,A -85,B 0,C 180,E1 -18246.329,E2 -18246.329} C_VEL
LIN {X 0,Y 273.032,Z 400.944,A -85,B 0,C 180,E1 -18246.915,E2 -18246.915} C_VEL
LIN {X 0,Y 271.082,Z 412.309,A -85,B 0,C 180,E1 -18248.52,E2 -18248.52} C_VEL
LIN {X 0,Y 269.491,Z 421.612,A -85,B 0,C 180,E1 -18250.184,E2 -18250.184} C_VEL
LIN {X 0,Y 267.695,Z 430.092,A -85,B 0,C 180,E1 -18252.033,E2 -18252.033} C_VEL
LIN {X 0,Y 265.807,Z 438.337,A -85,B 0,C 180,E1 -18254.276,E2 -18254.276} C_VEL
LIN {X 0,Y 264.572,Z 443.972,A -85,B 0,C 180,E1 -18256.169,E2 -18256.169} C_VEL
LIN {X 0,Y 263.297,Z 449.466,A -85,B 0,C 180,E1 -18258.453,E2 -18258.453} C_VEL
LIN {X 0,Y 262.352,Z 453.776,A -85,B 0,C 180,E1 -18260.752,E2 -18260.752} C_VEL
LIN {X 0,Y 261.727,Z 457.509,A -85,B 0,C 180,E1 -18263.487,E2 -18263.487} C_VEL
LIN {X 0,Y 261.442,Z 459.296,A -85,B 0,C 180,E1 -18265.375,E2 -18265.375} C_VEL
LIN {X 0,Y 261.282,Z 460.286,A -85,B 0,C 180,E1 -18266.917,E2 -18266.917} C_VEL
LIN {X 0,Y 261.138,Z 461.125,A -85,B 0,C 180,E1 -18270.001,E2 -18270.001} C_VEL
LIN {X 0,Y 261.172,Z 460.931,A -85,B 0,C 180,E1 -18271.543,E2 -18271.543} C_VEL
LIN {X 0,Y 261.279,Z 460.345,A -85,B 0,C 180,E1 -18273.084,E2 -18273.084} C_VEL
LIN {X 0,Y 261.661,Z 458.022,A -85,B 0,C 180,E1 -18276.168,E2 -18276.168} C_VEL
LIN {X 0,Y 262.158,Z 455.156,A -85,B 0,C 180,E1 -18278.479,E2 -18278.479} C_VEL
LIN {X 0,Y 262.895,Z 451.27,A -85,B 0,C 180,E1 -18280.786,E2 -18280.786} C_VEL
LIN {X 0,Y 264.043,Z 446.251,A -85,B 0,C 180,E1 -18283.076,E2 -18283.076} C_VEL
LIN {X 0,Y 265.423,Z 439.931,A -85,B 0,C 180,E1 -18285.355,E2 -18285.355} C_VEL
LIN {X 0,Y 267.328,Z 432.015,A -85,B 0,C 180,E1 -18287.598,E2 -18287.598} C_VEL
LIN {X 0,Y 269.047,Z 423.948,A -85,B 0,C 180,E1 -18289.455,E2 -18289.455} C_VEL
LIN {X 0,Y 270.806,Z 414.108,A -85,B 0,C 180,E1 -18291.305,E2 -18291.305} C_VEL
LIN {X 0,Y 272.785,Z 403.055,A -85,B 0,C 180,E1 -18292.93,E2 -18292.93} C_VEL
LIN {X 0,Y 273.001,Z 398.866,A -85,B 0,C 180,E1 -18293.497,E2 -18293.497} C_VEL
LIN {X 0,Y 271.373,Z 387.736,A -85,B 0,C 180,E1 -18294.983,E2 -18294.983} C_VEL
LIN {X 0,Y 269.121,Z 377.381,A -85,B 0,C 180,E1 -18296.194,E2 -18296.194} C_VEL
LIN {X 0,Y 265.349,Z 364.714,A -85,B 0,C 180,E1 -18297.493,E2 -18297.493} C_VEL
LIN {X 0,Y 262.825,Z 357.576,A -85,B 0,C 180,E1 -18298.145,E2 -18298.145} C_VEL
LIN {X 0,Y 262.73,Z 356.874,A -85,B 0,C 180,E1 -18298.187,E2 -18298.187} C_VEL
LIN {X 0,Y 263.119,Z 353.22,A -85,B 0,C 180,E1 -18302.29,E2 -18302.29} C_VEL
LIN {X 0,Y 263.324,Z 351.638,A -85,B 0,C 180,E1 -18304.169,E2 -18304.169} C_VEL
LIN {X 0,Y 263.325,Z 348.643,A -85,B 0,C 180,E1 -18307.869,E2 -18307.869} C_VEL
LIN {X 0,Y 263.17,Z 347.128,A -85,B 0,C 180,E1 -18309.861,E2 -18309.861} C_VEL
LIN {X 0,Y 263.124,Z 346.713,A -85,B 0,C 180,E1 -18311.893,E2 -18311.893} C_VEL
LIN {X 0,Y 263.098,Z 346.714,A -85,B 0,C 180,E1 -18316.156,E2 -18316.156} C_VEL
LIN {X 0,Y 263.089,Z 346.712,A -85,B 0,C 180,E1 -18320.776,E2 -18320.776} C_VEL
LIN {X 0,Y 263.159,Z 346.704,A -85,B 0,C 180,E1 -18324.017,E2 -18324.017} C_VEL
LIN {X 0,Y 263.127,Z 346.706,A -85,B 0,C 180,E1 -18327.711,E2 -18327.711} C_VEL
LIN {X 0,Y 263.147,Z 346.704,A -85,B 0,C 180,E1 -18331.805,E2 -18331.805} C_VEL
LIN {X 0,Y 263.188,Z 346.699,A -85,B 0,C 180,E1 -18335.218,E2 -18335.218} C_VEL
LIN {X 0,Y 263.262,Z 346.69,A -85,B 0,C 180,E1 -18339.693,E2 -18339.693} C_VEL
LIN {X 0,Y 263.35,Z 346.682,A -85,B 0,C 180,E1 -18344.522,E2 -18344.522} C_VEL
LIN {X 0,Y 263.372,Z 346.677,A -85,B 0,C 180,E1 -18349.234,E2 -18349.234} C_VEL
LIN {X 0,Y 263.572,Z 346.655,A -85,B 0,C 180,E1 -18352.338,E2 -18352.338} C_VEL
LIN {X 0,Y 263.746,Z 346.632,A -85,B 0,C 180,E1 -18358.473,E2 -18358.473} C_VEL
LIN {X 0,Y 263.745,Z 346.629,A -85,B 0,C 180,E1 -18361.527,E2 -18361.527} C_VEL
LIN {X 0,Y 263.557,Z 346.656,A -85,B 0,C 180,E1 -18367.662,E2 -18367.662} C_VEL
LIN {X 0,Y 263.353,Z 346.68,A -85,B 0,C 180,E1 -18370.766,E2 -18370.766} C_VEL
LIN {X 0,Y 263.343,Z 346.683,A -85,B 0,C 180,E1 -18375.478,E2 -18375.478} C_VEL
LIN {X 0,Y 263.262,Z 346.692,A -85,B 0,C 180,E1 -18380.307,E2 -18380.307} C_VEL
LIN {X 0,Y 263.117,Z 346.708,A -85,B 0,C 180,E1 -18382.729,E2 -18382.729} C_VEL
LIN {X 0,Y 262.452,Z 346.793,A -85,B 0,C 180,E1 -18384.006,E2 -18384.006} C_VEL
LIN {X 0,Y 259.595,Z 347.15,A -85,B 0,C 180,E1 -18386.087,E2 -18386.087} C_VEL
LIN {X 0,Y 257.17,Z 347.452,A -85,B 0,C 180,E1 -18387.779,E2 -18387.779} C_VEL
LIN {X 0,Y 256.135,Z 347.581,A -85,B 0,C 180,E1 -18389.092,E2 -18389.092} C_VEL
LIN {X 0,Y 256.053,Z 347.592,A -85,B 0,C 180,E1 -18389.537,E2 -18389.537} C_VEL
LIN {X 0,Y 256.065,Z 347.593,A -85,B 0,C 180,E1 -18393.293,E2 -18393.293} C_VEL
LIN {X 0,Y 256.109,Z 347.586,A -85,B 0,C 180,E1 -18397.269,E2 -18397.269} C_VEL
LIN {X 0,Y 256.094,Z 347.619,A -85,B 0,C 180,E1 -18399.465,E2 -18399.465} C_VEL
LIN {X 0,Y 256.617,Z 350.9,A -85,B 0,C 180,E1 -18403.21,E2 -18403.21} C_VEL
LIN {X 0,Y 257.365,Z 354.956,A -85,B 0,C 180,E1 -18407.502,E2 -18407.502} C_VEL
LIN {X 0,Y 257.784,Z 357.2,A -85,B 0,C 180,E1 -18409.762,E2 -18409.762} C_VEL
LIN {X 0,Y 257.931,Z 360.821,A -85,B 0,C 180,E1 -18413.17,E2 -18413.17} C_VEL
LIN {X 0,Y 257.684,Z 364,A -85,B 0,C 180,E1 -18416.006,E2 -18416.006} C_VEL
LIN {X 0,Y 256.692,Z 369.211,A -85,B 0,C 180,E1 -18420.473,E2 -18420.473} C_VEL
LIN {X 0,Y 256.558,Z 369.93,A -85,B 0,C 180,E1 -18421.081,E2 -18421.081} C_VEL
LIN {X 0,Y 260.233,Z 384.026,A -85,B 0,C 180,E1 -18422.295,E2 -18422.295} C_VEL
LIN {X 0,Y 262.624,Z 396.219,A -85,B 0,C 180,E1 -18423.55,E2 -18423.55} C_VEL
LIN {X 0,Y 263.988,Z 407.057,A -85,B 0,C 180,E1 -18424.845,E2 -18424.845} C_VEL
LIN {X 0,Y 264.719,Z 419.091,A -85,B 0,C 180,E1 -18426.532,E2 -18426.532} C_VEL
LIN {X 0,Y 264.488,Z 423.006,A -85,B 0,C 180,E1 -18427.131,E2 -18427.131} C_VEL
LIN {X 0,Y 262.438,Z 433.18,A -85,B 0,C 180,E1 -18428.806,E2 -18428.806} C_VEL
LIN {X 0,Y 260.489,Z 442.693,A -85,B 0,C 180,E1 -18430.787,E2 -18430.787} C_VEL
LIN {X 0,Y 258.547,Z 451.281,A -85,B 0,C 180,E1 -18433.009,E2 -18433.009} C_VEL
LIN {X 0,Y 256.961,Z 458.474,A -85,B 0,C 180,E1 -18435.345,E2 -18435.345} C_VEL
LIN {X 0,Y 255.848,Z 463.33,A -85,B 0,C 180,E1 -18437.305,E2 -18437.305} C_VEL
LIN {X 0,Y 254.975,Z 468.057,A -85,B 0,C 180,E1 -18439.679,E2 -18439.679} C_VEL
LIN {X 0,Y 254.375,Z 471.669,A -85,B 0,C 180,E1 -18442.059,E2 -18442.059} C_VEL
LIN {X 0,Y 254.022,Z 474.67,A -85,B 0,C 180,E1 -18444.881,E2 -18444.881} C_VEL
LIN {X 0,Y 253.987,Z 475.934,A -85,B 0,C 180,E1 -18446.827,E2 -18446.827} C_VEL
LIN {X 0,Y 254.015,Z 476.546,A -85,B 0,C 180,E1 -18448.414,E2 -18448.414} C_VEL
LIN {X 0,Y 254.032,Z 476.761,A -85,B 0,C 180,E1 -18449.999,E2 -18449.999} C_VEL
LIN {X 0,Y 254.015,Z 476.539,A -85,B 0,C 180,E1 -18451.585,E2 -18451.585} C_VEL
LIN {X 0,Y 253.987,Z 475.925,A -85,B 0,C 180,E1 -18453.172,E2 -18453.172} C_VEL
LIN {X 0,Y 254.021,Z 474.655,A -85,B 0,C 180,E1 -18455.118,E2 -18455.118} C_VEL
LIN {X 0,Y 254.372,Z 471.642,A -85,B 0,C 180,E1 -18457.94,E2 -18457.94} C_VEL
LIN {X 0,Y 254.975,Z 468.015,A -85,B 0,C 180,E1 -18460.32,E2 -18460.32} C_VEL
LIN {X 0,Y 255.847,Z 463.278,A -85,B 0,C 180,E1 -18462.694,E2 -18462.694} C_VEL
LIN {X 0,Y 257.463,Z 456.172,A -85,B 0,C 180,E1 -18465.434,E2 -18465.434} C_VEL
LIN {X 0,Y 259.238,Z 448.46,A -85,B 0,C 180,E1 -18467.756,E2 -18467.756} C_VEL
LIN {X 0,Y 261.217,Z 438.778,A -85,B 0,C 180,E1 -18470.06,E2 -18470.06} C_VEL
LIN {X 0,Y 263.266,Z 428.792,A -85,B 0,C 180,E1 -18471.945,E2 -18471.945} C_VEL
LIN {X 0,Y 264.709,Z 421.556,A -85,B 0,C 180,E1 -18473.054,E2 -18473.054} C_VEL
LIN {X 0,Y 264.215,Z 410.09,A -85,B 0,C 180,E1 -18474.736,E2 -18474.736} C_VEL
LIN {X 0,Y 262.921,Z 398.325,A -85,B 0,C 180,E1 -18476.192,E2 -18476.192} C_VEL
LIN {X 0,Y 260.583,Z 385.759,A -85,B 0,C 180,E1 -18477.511,E2 -18477.511} C_VEL
LIN {X 0,Y 257.133,Z 372.508,A -85,B 0,C 180,E1 -18478.693,E2 -18478.693} C_VEL
LIN {X 0,Y 256.565,Z 369.936,A -85,B 0,C 180,E1 -18478.883,E2 -18478.883} C_VEL
LIN {X 0,Y 257.498,Z 365.019,A -85,B 0,C 180,E1 -18483.082,E2 -18483.082} C_VEL
LIN {X 0,Y 257.889,Z 362.633,A -85,B 0,C 180,E1 -18485.158,E2 -18485.158} C_VEL
LIN {X 0,Y 257.956,Z 358.655,A -85,B 0,C 180,E1 -18488.801,E2 -18488.801} C_VEL
LIN {X 0,Y 257.415,Z 354.892,A -85,B 0,C 180,E1 -18492.51,E2 -18492.51} C_VEL
LIN {X 0,Y 256.638,Z 350.868,A -85,B 0,C 180,E1 -18496.794,E2 -18496.794} C_VEL
LIN {X 0,Y 256.058,Z 347.59,A -85,B 0,C 180,E1 -18500.528,E2 -18500.528} C_VEL
LIN {X 0,Y 256.12,Z 347.581,A -85,B 0,C 180,E1 -18502.866,E2 -18502.866} C_VEL
LIN {X 0,Y 256.06,Z 347.591,A -85,B 0,C 180,E1 -18506.706,E2 -18506.706} C_VEL
LIN {X 0,Y 256.048,Z 347.594,A -85,B 0,C 180,E1 -18510.392,E2 -18510.392} C_VEL
LIN {X 0,Y 256.126,Z 347.582,A -85,B 0,C 180,E1 -18514.888,E2 -18514.888} C_VEL
LIN {X 0,Y 256.155,Z 347.576,A -85,B 0,C 180,E1 -18519.104,E2 -18519.104} C_VEL
LIN {X 0,Y 256.287,Z 347.562,A -85,B 0,C 180,E1 -18524.084,E2 -18524.084} C_VEL
LIN {X 0,Y 256.302,Z 347.556,A -85,B 0,C 180,E1 -18528.934,E2 -18528.934} C_VEL
LIN {X 0,Y 256.533,Z 347.531,A -85,B 0,C 180,E1 -18532.127,E2 -18532.127} C_VEL
LIN {X 0,Y 256.704,Z 347.507,A -85,B 0,C 180,E1 -18538.431,E2 -18538.431} C_VEL
LIN {X 0,Y 256.704,Z 347.51,A -85,B 0,C 180,E1 -18541.569,E2 -18541.569} C_VEL
LIN {X 0,Y 256.533,Z 347.528,A -85,B 0,C 180,E1 -18547.873,E2 -18547.873} C_VEL
LIN {X 0,Y 256.302,Z 347.559,A -85,B 0,C 180,E1 -18551.066,E2 -18551.066} C_VEL
LIN {X 0,Y 256.293,Z 347.559,A -85,B 0,C 180,E1 -18555.916,E2 -18555.916} C_VEL
LIN {X 0,Y 256.157,Z 347.578,A -85,B 0,C 180,E1 -18560.896,E2 -18560.896} C_VEL
LIN {X 0,Y 256.127,Z 347.582,A -85,B 0,C 180,E1 -18565.113,E2 -18565.113} C_VEL
LIN {X 0,Y 256.048,Z 347.59,A -85,B 0,C 180,E1 -18569.608,E2 -18569.608} C_VEL
LIN {X 0,Y 256.06,Z 347.589,A -85,B 0,C 180,E1 -18573.294,E2 -18573.294} C_VEL
LIN {X 0,Y 256.106,Z 347.583,A -85,B 0,C 180,E1 -18577.271,E2 -18577.271} C_VEL
LIN {X 0,Y 256.013,Z 347.593,A -85,B 0,C 180,E1 -18581.212,E2 -18581.212} C_VEL
LIN {X 0,Y 256.052,Z 347.59,A -85,B 0,C 180,E1 -18585.532,E2 -18585.532} C_VEL
LIN {X 0,Y 256.073,Z 347.589,A -85,B 0,C 180,E1 -18588.802,E2 -18588.802} C_VEL
LIN {X 0,Y 256.253,Z 348.747,A -85,B 0,C 180,E1 -18590.893,E2 -18590.893} C_VEL
LIN {X 0,Y 256.35,Z 350.266,A -85,B 0,C 180,E1 -18592.906,E2 -18592.906} C_VEL
LIN {X 0,Y 256.313,Z 352.194,A -85,B 0,C 180,E1 -18595.345,E2 -18595.345} C_VEL
LIN {X 0,Y 256.033,Z 354.882,A -85,B 0,C 180,E1 -18598.566,E2 -18598.566} C_VEL
LIN {X 0,Y 255.786,Z 357.072,A -85,B 0,C 180,E1 -18601.085,E2 -18601.085} C_VEL
LIN {X 0,Y 257.75,Z 362.937,A -85,B 0,C 180,E1 -18601.633,E2 -18601.633} C_VEL
LIN {X 0,Y 261.336,Z 374.1,A -85,B 0,C 180,E1 -18602.796,E2 -18602.796} C_VEL
LIN {X 0,Y 264.143,Z 385.756,A -85,B 0,C 180,E1 -18604.172,E2 -18604.172} C_VEL
LIN {X 0,Y 265.857,Z 396.163,A -85,B 0,C 180,E1 -18605.567,E2 -18605.567} C_VEL
LIN {X 0,Y 266.422,Z 401.363,A -85,B 0,C 180,E1 -18606.337,E2 -18606.337} C_VEL
LIN {X 0,Y 264.504,Z 412.528,A -85,B 0,C 180,E1 -18607.958,E2 -18607.958} C_VEL
LIN {X 0,Y 262.81,Z 421.831,A -85,B 0,C 180,E1 -18609.658,E2 -18609.658} C_VEL
LIN {X 0,Y 260.96,Z 430.31,A -85,B 0,C 180,E1 -18611.553,E2 -18611.553} C_VEL
LIN {X 0,Y 258.985,Z 438.554,A -85,B 0,C 180,E1 -18613.851,E2 -18613.851} C_VEL
LIN {X 0,Y 257.678,Z 444.189,A -85,B 0,C 180,E1 -18615.791,E2 -18615.791} C_VEL
LIN {X 0,Y 256.349,Z 449.683,A -85,B 0,C 180,E1 -18618.135,E2 -18618.135} C_VEL
LIN {X 0,Y 255.351,Z 453.993,A -85,B 0,C 180,E1 -18620.496,E2 -18620.496} C_VEL
LIN {X 0,Y 254.645,Z 457.944,A -85,B 0,C 180,E1 -18623.502,E2 -18623.502} C_VEL
LIN {X 0,Y 254.359,Z 459.512,A -85,B 0,C 180,E1 -18625.246,E2 -18625.246} C_VEL
LIN {X 0,Y 254.201,Z 460.502,A -85,B 0,C 180,E1 -18626.831,E2 -18626.831} C_VEL
LIN {X 0,Y 254.103,Z 461.111,A -85,B 0,C 180,E1 -18628.416,E2 -18628.416} C_VEL
LIN {X 0,Y 254.066,Z 461.34,A -85,B 0,C 180,E1 -18630.001,E2 -18630.001} C_VEL
LIN {X 0,Y 254.103,Z 461.146,A -85,B 0,C 180,E1 -18631.586,E2 -18631.586} C_VEL
LIN {X 0,Y 254.196,Z 460.56,A -85,B 0,C 180,E1 -18633.17,E2 -18633.17} C_VEL
LIN {X 0,Y 254.606,Z 458.236,A -85,B 0,C 180,E1 -18636.34,E2 -18636.34} C_VEL
LIN {X 0,Y 255.128,Z 455.371,A -85,B 0,C 180,E1 -18638.715,E2 -18638.715} C_VEL
LIN {X 0,Y 255.931,Z 451.484,A -85,B 0,C 180,E1 -18641.083,E2 -18641.083} C_VEL
LIN {X 0,Y 257.13,Z 446.465,A -85,B 0,C 180,E1 -18643.435,E2 -18643.435} C_VEL
LIN {X 0,Y 258.581,Z 440.145,A -85,B 0,C 180,E1 -18645.771,E2 -18645.771} C_VEL
LIN {X 0,Y 260.556,Z 432.229,A -85,B 0,C 180,E1 -18648.071,E2 -18648.071} C_VEL
LIN {X 0,Y 262.357,Z 424.161,A -85,B 0,C 180,E1 -18649.971,E2 -18649.971} C_VEL
LIN {X 0,Y 264.206,Z 414.319,A -85,B 0,C 180,E1 -18651.864,E2 -18651.864} C_VEL
LIN {X 0,Y 266.254,Z 403.358,A -85,B 0,C 180,E1 -18653.512,E2 -18653.512} C_VEL
LIN {X 0,Y 266.308,Z 399.485,A -85,B 0,C 180,E1 -18654.07,E2 -18654.07} C_VEL
LIN {X 0,Y 264.8,Z 389.087,A -85,B 0,C 180,E1 -18655.526,E2 -18655.526} C_VEL
LIN {X 0,Y 262.179,Z 377.356,A -85,B 0,C 180,E1 -18656.963,E2 -18656.963} C_VEL
LIN {X 0,Y 258.684,Z 365.684,A -85,B 0,C 180,E1 -18658.219,E2 -18658.219} C_VEL
LIN {X 0,Y 255.864,Z 357.757,A -85,B 0,C 180,E1 -18658.984,E2 -18658.984} C_VEL
LIN {X 0,Y 255.764,Z 357.085,A -85,B 0,C 180,E1 -18659.037,E2 -18659.037} C_VEL
LIN {X 0,Y 256.035,Z 354.784,A -85,B 0,C 180,E1 -18661.686,E2 -18661.686} C_VEL
LIN {X 0,Y 256.3,Z 351.906,A -85,B 0,C 180,E1 -18665.159,E2 -18665.159} C_VEL
LIN {X 0,Y 256.356,Z 350.182,A -85,B 0,C 180,E1 -18667.341,E2 -18667.341} C_VEL
LIN {X 0,Y 256.175,Z 348.35,A -85,B 0,C 180,E1 -18669.81,E2 -18669.81} C_VEL
LIN {X 0,Y 256.064,Z 347.593,A -85,B 0,C 180,E1 -18671.202,E2 -18671.202} C_VEL
LIN {X 0,Y 256.037,Z 347.595,A -85,B 0,C 180,E1 -18675.535,E2 -18675.535} C_VEL
LIN {X 0,Y 256.008,Z 347.595,A -85,B 0,C 180,E1 -18678.787,E2 -18678.787} C_VEL
LIN {X 0,Y 256.1,Z 347.583,A -85,B 0,C 180,E1 -18682.862,E2 -18682.862} C_VEL
LIN {X 0,Y 256.066,Z 347.588,A -85,B 0,C 180,E1 -18686.707,E2 -18686.707} C_VEL
LIN {X 0,Y 256.054,Z 347.588,A -85,B 0,C 180,E1 -18690.393,E2 -18690.393} C_VEL
LIN {X 0,Y 256.132,Z 347.578,A -85,B 0,C 180,E1 -18694.888,E2 -18694.888} C_VEL
LIN {X 0,Y 256.161,Z 347.578,A -85,B 0,C 180,E1 -18699.104,E2 -18699.104} C_VEL
LIN {X 0,Y 256.299,Z 347.558,A -85,B 0,C 180,E1 -18704.085,E2 -18704.085} C_VEL
LIN {X 0,Y 256.308,Z 347.559,A -85,B 0,C 180,E1 -18708.934,E2 -18708.934} C_VEL
LIN {X 0,Y 256.539,Z 347.529,A -85,B 0,C 180,E1 -18712.127,E2 -18712.127} C_VEL
LIN {X 0,Y 256.709,Z 347.509,A -85,B 0,C 180,E1 -18718.431,E2 -18718.431} C_VEL
LIN {X 0,Y 256.709,Z 347.506,A -85,B 0,C 180,E1 -18721.569,E2 -18721.569} C_VEL
LIN {X 0,Y 256.479,Z 347.538,A -85,B 0,C 180,E1 -18726.293,E2 -18726.293} C_VEL
LIN {X 0,Y 256.426,Z 347.543,A -85,B 0,C 180,E1 -18729.465,E2 -18729.465} C_VEL
LIN {X 0,Y 256.25,Z 347.568,A -85,B 0,C 180,E1 -18734.29,E2 -18734.29} C_VEL
LIN {X 0,Y 256.209,Z 347.573,A -85,B 0,C 180,E1 -18737.562,E2 -18737.562} C_VEL
LIN {X 0,Y 256.152,Z 347.578,A -85,B 0,C 180,E1 -18741.117,E2 -18741.117} C_VEL
LIN {X 0,Y 256.132,Z 347.58,A -85,B 0,C 180,E1 -18745.112,E2 -18745.112} C_VEL
LIN {X 0,Y 256.053,Z 347.592,A -85,B 0,C 180,E1 -18749.537,E2 -18749.537} C_VEL
LIN {X 0,Y 255.4,Z 347.68,A -85,B 0,C 180,E1 -18750.849,E2 -18750.849} C_VEL
LIN {X 0,Y 252.575,Z 348.036,A -85,B 0,C 180,E1 -18752.99,E2 -18752.99} C_VEL
LIN {X 0,Y 250.162,Z 348.333,A -85,B 0,C 180,E1 -18754.732,E2 -18754.732} C_VEL
LIN {X 0,Y 249.112,Z 348.457,A -85,B 0,C 180,E1 -18756.082,E2 -18756.082} C_VEL
LIN {X 0,Y 249.018,Z 348.467,A -85,B 0,C 180,E1 -18756.54,E2 -18756.54} C_VEL
LIN {X 0,Y 249.032,Z 348.595,A -85,B 0,C 180,E1 -18758.897,E2 -18758.897} C_VEL
LIN {X 0,Y 249.604,Z 351.992,A -85,B 0,C 180,E1 -18762.94,E2 -18762.94} C_VEL
LIN {X 0,Y 250.415,Z 356.314,A -85,B 0,C 180,E1 -18767.657,E2 -18767.657} C_VEL
LIN {X 0,Y 250.799,Z 358.461,A -85,B 0,C 180,E1 -18769.871,E2 -18769.871} C_VEL
LIN {X 0,Y 250.917,Z 361.654,A -85,B 0,C 180,E1 -18772.972,E2 -18772.972} C_VEL
LIN {X 0,Y 250.672,Z 364.833,A -85,B 0,C 180,E1 -18775.894,E2 -18775.894} C_VEL
LIN {X 0,Y 249.683,Z 369.727,A -85,B 0,C 180,E1 -18780.214,E2 -18780.214} C_VEL
LIN {X 0,Y 251.342,Z 375.805,A -85,B 0,C 180,E1 -18780.723,E2 -18780.723} C_VEL
LIN {X 0,Y 254.58,Z 388.924,A -85,B 0,C 180,E1 -18782.011,E2 -18782.011} C_VEL
LIN {X 0,Y 256.595,Z 400.781,A -85,B 0,C 180,E1 -18783.367,E2 -18783.367} C_VEL
LIN {X 0,Y 257.665,Z 411.993,A -85,B 0,C 180,E1 -18784.851,E2 -18784.851} C_VEL
LIN {X 0,Y 257.984,Z 421.492,A -85,B 0,C 180,E1 -18786.308,E2 -18786.308} C_VEL
LIN {X 0,Y 256.732,Z 428.71,A -85,B 0,C 180,E1 -18787.465,E2 -18787.465} C_VEL
LIN {X 0,Y 254.524,Z 438.847,A -85,B 0,C 180,E1 -18789.429,E2 -18789.429} C_VEL
LIN {X 0,Y 252.467,Z 448.355,A -85,B 0,C 180,E1 -18791.756,E2 -18791.756} C_VEL
LIN {X 0,Y 250.608,Z 456.021,A -85,B 0,C 180,E1 -18794.131,E2 -18794.131} C_VEL
LIN {X 0,Y 248.885,Z 463.115,A -85,B 0,C 180,E1 -18796.944,E2 -18796.944} C_VEL
LIN {X 0,Y 247.95,Z 467.841,A -85,B 0,C 180,E1 -18799.383,E2 -18799.383} C_VEL
LIN {X 0,Y 247.342,Z 471.455,A -85,B 0,C 180,E1 -18801.832,E2 -18801.832} C_VEL
LIN {X 0,Y 247.075,Z 473.319,A -85,B 0,C 180,E1 -18803.466,E2 -18803.466} C_VEL
LIN {X 0,Y 246.923,Z 474.718,A -85,B 0,C 180,E1 -18805.101,E2 -18805.101} C_VEL
LIN {X 0,Y 246.889,Z 475.719,A -85,B 0,C 180,E1 -18806.736,E2 -18806.736} C_VEL
LIN {X 0,Y 246.924,Z 476.33,A -85,B 0,C 180,E1 -18808.368,E2 -18808.368} C_VEL
LIN {X 0,Y 246.962,Z 476.546,A -85,B 0,C 180,E1 -18809.999,E2 -18809.999} C_VEL
LIN {X 0,Y 246.924,Z 476.324,A -85,B 0,C 180,E1 -18811.63,E2 -18811.63} C_VEL
LIN {X 0,Y 246.889,Z 475.709,A -85,B 0,C 180,E1 -18813.263,E2 -18813.263} C_VEL
LIN {X 0,Y 246.944,Z 474.59,A -85,B 0,C 180,E1 -18815.063,E2 -18815.063} C_VEL
LIN {X 0,Y 247.074,Z 473.299,A -85,B 0,C 180,E1 -18816.532,E2 -18816.532} C_VEL
LIN {X 0,Y 247.517,Z 470.35,A -85,B 0,C 180,E1 -18818.984,E2 -18818.984} C_VEL
LIN {X 0,Y 248.237,Z 466.362,A -85,B 0,C 180,E1 -18821.43,E2 -18821.43} C_VEL
LIN {X 0,Y 249.535,Z 460.235,A -85,B 0,C 180,E1 -18824.266,E2 -18824.266} C_VEL
LIN {X 0,Y 251.2,Z 453.551,A -85,B 0,C 180,E1 -18826.664,E2 -18826.664} C_VEL
LIN {X 0,Y 253.229,Z 444.884,A -85,B 0,C 180,E1 -18829.135,E2 -18829.135} C_VEL
LIN {X 0,Y 254.92,Z 436.753,A -85,B 0,C 180,E1 -18831.001,E2 -18831.001} C_VEL
LIN {X 0,Y 257.195,Z 426.255,A -85,B 0,C 180,E1 -18832.915,E2 -18832.915} C_VEL
LIN {X 0,Y 257.94,Z 421.328,A -85,B 0,C 180,E1 -18833.695,E2 -18833.695} C_VEL
LIN {X 0,Y 257.515,Z 410.9,A -85,B 0,C 180,E1 -18835.283,E2 -18835.283} C_VEL
LIN {X 0,Y 256.322,Z 399.081,A -85,B 0,C 180,E1 -18836.818,E2 -18836.818} C_VEL
LIN {X 0,Y 254.116,Z 386.839,A -85,B 0,C 180,E1 -18838.177,E2 -18838.177} C_VEL
LIN {X 0,Y 250.553,Z 373.029,A -85,B 0,C 180,E1 -18839.481,E2 -18839.481} C_VEL
LIN {X 0,Y 249.684,Z 369.661,A -85,B 0,C 180,E1 -18839.812,E2 -18839.812} C_VEL
LIN {X 0,Y 250.669,Z 364.797,A -85,B 0,C 180,E1 -18844.105,E2 -18844.105} C_VEL
LIN {X 0,Y 250.948,Z 361.626,A -85,B 0,C 180,E1 -18847.021,E2 -18847.021} C_VEL
LIN {X 0,Y 250.807,Z 358.425,A -85,B 0,C 180,E1 -18850.126,E2 -18850.126} C_VEL
LIN {X 0,Y 250.319,Z 355.527,A -85,B 0,C 180,E1 -18853.115,E2 -18853.115} C_VEL
LIN {X 0,Y 249.554,Z 351.592,A -85,B 0,C 180,E1 -18857.476,E2 -18857.476} C_VEL
LIN {X 0,Y 249.012,Z 348.471,A -85,B 0,C 180,E1 -18861.358,E2 -18861.358} C_VEL
LIN {X 0,Y 249.037,Z 348.464,A -85,B 0,C 180,E1 -18865.638,E2 -18865.638} C_VEL
LIN {X 0,Y 248.996,Z 348.469,A -85,B 0,C 180,E1 -18869.465,E2 -18869.465} C_VEL
LIN {X 0,Y 249.028,Z 348.466,A -85,B 0,C 180,E1 -18873.157,E2 -18873.157} C_VEL
LIN {X 0,Y 249.049,Z 348.463,A -85,B 0,C 180,E1 -18876.73,E2 -18876.73} C_VEL
LIN {X 0,Y 249.102,Z 348.456,A -85,B 0,C 180,E1 -18880.211,E2 -18880.211} C_VEL
LIN {X 0,Y 249.236,Z 348.439,A -85,B 0,C 180,E1 -18883.621,E2 -18883.621} C_VEL
LIN {X 0,Y 249.245,Z 348.436,A -85,B 0,C 180,E1 -18888.616,E2 -18888.616} C_VEL
LIN {X 0,Y 249.475,Z 348.41,A -85,B 0,C 180,E1 -18891.903,E2 -18891.903} C_VEL
LIN {X 0,Y 249.43,Z 348.412,A -85,B 0,C 180,E1 -18896.77,E2 -18896.77} C_VEL
LIN {X 0,Y 249.667,Z 348.384,A -85,B 0,C 180,E1 -18898.387,E2 -18898.387} C_VEL
LIN {X 0,Y 249.666,Z 348.387,A -85,B 0,C 180,E1 -18901.613,E2 -18901.613} C_VEL
LIN {X 0,Y 249.445,Z 348.41,A -85,B 0,C 180,E1 -18906.731,E2 -18906.731} C_VEL
LIN {X 0,Y 249.418,Z 348.417,A -85,B 0,C 180,E1 -18909.734,E2 -18909.734} C_VEL
LIN {X 0,Y 249.198,Z 348.441,A -85,B 0,C 180,E1 -18914.704,E2 -18914.704} C_VEL
LIN {X 0,Y 249.133,Z 348.451,A -85,B 0,C 180,E1 -18918.078,E2 -18918.078} C_VEL
LIN {X 0,Y 249.078,Z 348.458,A -85,B 0,C 180,E1 -18921.519,E2 -18921.519} C_VEL
LIN {X 0,Y 249.079,Z 348.459,A -85,B 0,C 180,E1 -18925.461,E2 -18925.461} C_VEL
LIN {X 0,Y 249.031,Z 348.466,A -85,B 0,C 180,E1 -18928.975,E2 -18928.975} C_VEL
LIN {X 0,Y 249.022,Z 348.467,A -85,B 0,C 180,E1 -18932.427,E2 -18932.427} C_VEL
LIN {X 0,Y 249.04,Z 348.464,A -85,B 0,C 180,E1 -18936.344,E2 -18936.344} C_VEL
LIN {X 0,Y 248.974,Z 348.472,A -85,B 0,C 180,E1 -18940.485,E2 -18940.485} C_VEL
LIN {X 0,Y 248.988,Z 348.47,A -85,B 0,C 180,E1 -18944.883,E2 -18944.883} C_VEL
LIN {X 0,Y 249.024,Z 348.467,A -85,B 0,C 180,E1 -18947.366,E2 -18947.366} C_VEL
LIN {X 0,Y 249.087,Z 349.042,A -85,B 0,C 180,E1 -18949.624,E2 -18949.624} C_VEL
LIN {X 0,Y 249.295,Z 350.827,A -85,B 0,C 180,E1 -18952.126,E2 -18952.126} C_VEL
LIN {X 0,Y 249.239,Z 353.557,A -85,B 0,C 180,E1 -18955.672,E2 -18955.672} C_VEL
LIN {X 0,Y 248.827,Z 357.337,A -85,B 0,C 180,E1 -18960.22,E2 -18960.22} C_VEL
LIN {X 0,Y 249.869,Z 360.526,A -85,B 0,C 180,E1 -18960.514,E2 -18960.514} C_VEL
LIN {X 0,Y 254.067,Z 372.887,A -85,B 0,C 180,E1 -18961.839,E2 -18961.839} C_VEL
LIN {X 0,Y 256.797,Z 383.52,A -85,B 0,C 180,E1 -18963.116,E2 -18963.116} C_VEL
LIN {X 0,Y 258.883,Z 394.512,A -85,B 0,C 180,E1 -18964.611,E2 -18964.611} C_VEL
LIN {X 0,Y 259.773,Z 402.906,A -85,B 0,C 180,E1 -18965.89,E2 -18965.89} C_VEL
LIN {X 0,Y 257.711,Z 413.901,A -85,B 0,C 180,E1 -18967.556,E2 -18967.556} C_VEL
LIN {X 0,Y 255.734,Z 423.854,A -85,B 0,C 180,E1 -18969.49,E2 -18969.49} C_VEL
LIN {X 0,Y 253.866,Z 432.007,A -85,B 0,C 180,E1 -18971.437,E2 -18971.437} C_VEL
LIN {X 0,Y 251.82,Z 439.998,A -85,B 0,C 180,E1 -18973.795,E2 -18973.795} C_VEL
LIN {X 0,Y 250.29,Z 446.404,A -85,B 0,C 180,E1 -18976.193,E2 -18976.193} C_VEL
LIN {X 0,Y 249.018,Z 451.485,A -85,B 0,C 180,E1 -18978.607,E2 -18978.607} C_VEL
LIN {X 0,Y 248.076,Z 455.429,A -85,B 0,C 180,E1 -18981.037,E2 -18981.037} C_VEL
LIN {X 0,Y 247.521,Z 458.459,A -85,B 0,C 180,E1 -18983.606,E2 -18983.606} C_VEL
LIN {X 0,Y 247.122,Z 460.717,A -85,B 0,C 180,E1 -18986.74,E2 -18986.74} C_VEL
LIN {X 0,Y 247.036,Z 461.325,A -85,B 0,C 180,E1 -18988.371,E2 -18988.371} C_VEL
LIN {X 0,Y 246.995,Z 461.554,A -85,B 0,C 180,E1 -18990.001,E2 -18990.001} C_VEL
LIN {X 0,Y 247.035,Z 461.36,A -85,B 0,C 180,E1 -18991.631,E2 -18991.631} C_VEL
LIN {X 0,Y 247.116,Z 460.775,A -85,B 0,C 180,E1 -18993.261,E2 -18993.261} C_VEL
LIN {X 0,Y 247.547,Z 458.451,A -85,B 0,C 180,E1 -18996.521,E2 -18996.521} C_VEL
LIN {X 0,Y 248.1,Z 455.586,A -85,B 0,C 180,E1 -18998.964,E2 -18998.964} C_VEL
LIN {X 0,Y 248.953,Z 451.698,A -85,B 0,C 180,E1 -19001.398,E2 -19001.398} C_VEL
LIN {X 0,Y 250.214,Z 446.679,A -85,B 0,C 180,E1 -19003.813,E2 -19003.813} C_VEL
LIN {X 0,Y 251.757,Z 440.358,A -85,B 0,C 180,E1 -19006.21,E2 -19006.21} C_VEL
LIN {X 0,Y 253.796,Z 432.442,A -85,B 0,C 180,E1 -19008.57,E2 -19008.57} C_VEL
LIN {X 0,Y 255.677,Z 424.418,A -85,B 0,C 180,E1 -19010.506,E2 -19010.506} C_VEL
LIN {X 0,Y 257.398,Z 415.598,A -85,B 0,C 180,E1 -19012.262,E2 -19012.262} C_VEL
LIN {X 0,Y 259.543,Z 404.833,A -85,B 0,C 180,E1 -19013.965,E2 -19013.965} C_VEL
LIN {X 0,Y 259.73,Z 401.295,A -85,B 0,C 180,E1 -19014.482,E2 -19014.482} C_VEL
LIN {X 0,Y 258.24,Z 390.432,A -85,B 0,C 180,E1 -19016.091,E2 -19016.091} C_VEL
LIN {X 0,Y 255.726,Z 378.89,A -85,B 0,C 180,E1 -19017.588,E2 -19017.588} C_VEL
LIN {X 0,Y 252.185,Z 366.886,A -85,B 0,C 180,E1 -19018.952,E2 -19018.952} C_VEL
LIN {X 0,Y 248.868,Z 357.774,A -85,B 0,C 180,E1 -19019.889,E2 -19019.889} C_VEL
LIN {X 0,Y 248.831,Z 357.269,A -85,B 0,C 180,E1 -19019.972,E2 -19019.972} C_VEL
LIN {X 0,Y 249.227,Z 353.669,A -85,B 0,C 180,E1 -19024.332,E2 -19024.332} C_VEL
LIN {X 0,Y 249.3,Z 350.948,A -85,B 0,C 180,E1 -19027.875,E2 -19027.875} C_VEL
LIN {X 0,Y 249.091,Z 349.097,A -85,B 0,C 180,E1 -19030.461,E2 -19030.461} C_VEL
LIN {X 0,Y 249.002,Z 348.472,A -85,B 0,C 180,E1 -19032.79,E2 -19032.79} C_VEL
LIN {X 0,Y 248.983,Z 348.472,A -85,B 0,C 180,E1 -19037.355,E2 -19037.355} C_VEL
LIN {X 0,Y 249.039,Z 348.462,A -85,B 0,C 180,E1 -19042.202,E2 -19042.202} C_VEL
LIN {X 0,Y 249.043,Z 348.464,A -85,B 0,C 180,E1 -19045.639,E2 -19045.639} C_VEL
LIN {X 0,Y 249.001,Z 348.469,A -85,B 0,C 180,E1 -19049.466,E2 -19049.466} C_VEL
LIN {X 0,Y 249.034,Z 348.466,A -85,B 0,C 180,E1 -19053.157,E2 -19053.157} C_VEL
LIN {X 0,Y 249.055,Z 348.462,A -85,B 0,C 180,E1 -19056.73,E2 -19056.73} C_VEL
LIN {X 0,Y 249.108,Z 348.454,A -85,B 0,C 180,E1 -19060.211,E2 -19060.211} C_VEL
LIN {X 0,Y 249.242,Z 348.437,A -85,B 0,C 180,E1 -19063.622,E2 -19063.622} C_VEL
LIN {X 0,Y 249.252,Z 348.438,A -85,B 0,C 180,E1 -19068.616,E2 -19068.616} C_VEL
LIN {X 0,Y 249.481,Z 348.408,A -85,B 0,C 180,E1 -19071.903,E2 -19071.903} C_VEL
LIN {X 0,Y 249.433,Z 348.415,A -85,B 0,C 180,E1 -19076.769,E2 -19076.769} C_VEL
LIN {X 0,Y 249.671,Z 348.385,A -85,B 0,C 180,E1 -19078.387,E2 -19078.387} C_VEL
LIN {X 0,Y 249.671,Z 348.383,A -85,B 0,C 180,E1 -19081.613,E2 -19081.613} C_VEL
LIN {X 0,Y 249.452,Z 348.414,A -85,B 0,C 180,E1 -19086.471,E2 -19086.471} C_VEL
LIN {X 0,Y 249.343,Z 348.427,A -85,B 0,C 180,E1 -19089.736,E2 -19089.736} C_VEL
LIN {X 0,Y 249.2,Z 348.444,A -85,B 0,C 180,E1 -19094.704,E2 -19094.704} C_VEL
LIN {X 0,Y 249.138,Z 348.453,A -85,B 0,C 180,E1 -19098.077,E2 -19098.077} C_VEL
LIN {X 0,Y 249.083,Z 348.46,A -85,B 0,C 180,E1 -19101.519,E2 -19101.519} C_VEL
LIN {X 0,Y 249.084,Z 348.46,A -85,B 0,C 180,E1 -19105.46,E2 -19105.46} C_VEL
LIN {X 0,Y 249.002,Z 348.467,A -85,B 0,C 180,E1 -19109.522,E2 -19109.522} C_VEL
LIN {X 0,Y 249.026,Z 348.467,A -85,B 0,C 180,E1 -19112.426,E2 -19112.426} C_VEL
LIN {X 0,Y 249.018,Z 348.467,A -85,B 0,C 180,E1 -19116.54,E2 -19116.54} C_VEL
LIN {X 0,Y 248.368,Z 348.8,A -85,B 0,C 180,E1 -19117.888,E2 -19117.888} C_VEL
LIN {X 0,Y 246.894,Z 349.654,A -85,B 0,C 180,E1 -19119.205,E2 -19119.205} C_VEL
LIN {X 0,Y 243.556,Z 352.198,A -85,B 0,C 180,E1 -19121.835,E2 -19121.835} C_VEL
LIN {X 0,Y 242.733,Z 353.546,A -85,B 0,C 180,E1 -19123.197,E2 -19123.197} C_VEL
LIN {X 0,Y 242.721,Z 353.957,A -85,B 0,C 180,E1 -19123.658,E2 -19123.658} C_VEL
LIN {X 0,Y 243.591,Z 358.404,A -85,B 0,C 180,E1 -19128.603,E2 -19128.603} C_VEL
LIN {X 0,Y 243.834,Z 360.812,A -85,B 0,C 180,E1 -19131.098,E2 -19131.098} C_VEL
LIN {X 0,Y 243.83,Z 363.584,A -85,B 0,C 180,E1 -19133.809,E2 -19133.809} C_VEL
LIN {X 0,Y 243.358,Z 366.853,A -85,B 0,C 180,E1 -19136.877,E2 -19136.877} C_VEL
LIN {X 0,Y 242.828,Z 369.467,A -85,B 0,C 180,E1 -19139.266,E2 -19139.266} C_VEL
LIN {X 0,Y 244.45,Z 375.458,A -85,B 0,C 180,E1 -19139.807,E2 -19139.807} C_VEL
LIN {X 0,Y 247.544,Z 387.568,A -85,B 0,C 180,E1 -19141.044,E2 -19141.044} C_VEL
LIN {X 0,Y 249.601,Z 398.893,A -85,B 0,C 180,E1 -19142.371,E2 -19142.371} C_VEL
LIN {X 0,Y 250.844,Z 410.474,A -85,B 0,C 180,E1 -19143.936,E2 -19143.936} C_VEL
LIN {X 0,Y 251.266,Z 421.273,A -85,B 0,C 180,E1 -19145.634,E2 -19145.634} C_VEL
LIN {X 0,Y 250.947,Z 425.016,A -85,B 0,C 180,E1 -19146.26,E2 -19146.26} C_VEL
LIN {X 0,Y 248.747,Z 434.711,A -85,B 0,C 180,E1 -19148.015,E2 -19148.015} C_VEL
LIN {X 0,Y 246.783,Z 443.554,A -85,B 0,C 180,E1 -19150.017,E2 -19150.017} C_VEL
LIN {X 0,Y 244.966,Z 450.853,A -85,B 0,C 180,E1 -19152.036,E2 -19152.036} C_VEL
LIN {X 0,Y 243.171,Z 458.044,A -85,B 0,C 180,E1 -19154.494,E2 -19154.494} C_VEL
LIN {X 0,Y 241.936,Z 462.9,A -85,B 0,C 180,E1 -19156.562,E2 -19156.562} C_VEL
LIN {X 0,Y 240.942,Z 467.626,A -85,B 0,C 180,E1 -19159.07,E2 -19159.07} C_VEL
LIN {X 0,Y 240.282,Z 471.239,A -85,B 0,C 180,E1 -19161.59,E2 -19161.59} C_VEL
LIN {X 0,Y 240,Z 473.103,A -85,B 0,C 180,E1 -19163.273,E2 -19163.273} C_VEL
LIN {X 0,Y 239.837,Z 474.585,A -85,B 0,C 180,E1 -19165.078,E2 -19165.078} C_VEL
LIN {X 0,Y 239.835,Z 476.115,A -85,B 0,C 180,E1 -19168.32,E2 -19168.32} C_VEL
LIN {X 0,Y 239.872,Z 476.331,A -85,B 0,C 180,E1 -19169.999,E2 -19169.999} C_VEL
LIN {X 0,Y 239.835,Z 476.109,A -85,B 0,C 180,E1 -19171.678,E2 -19171.678} C_VEL
LIN {X 0,Y 239.837,Z 474.571,A -85,B 0,C 180,E1 -19174.921,E2 -19174.921} C_VEL
LIN {X 0,Y 239.999,Z 473.082,A -85,B 0,C 180,E1 -19176.726,E2 -19176.726} C_VEL
LIN {X 0,Y 240.468,Z 470.132,A -85,B 0,C 180,E1 -19179.249,E2 -19179.249} C_VEL
LIN {X 0,Y 241.255,Z 466.144,A -85,B 0,C 180,E1 -19181.765,E2 -19181.765} C_VEL
LIN {X 0,Y 242.647,Z 460.017,A -85,B 0,C 180,E1 -19184.68,E2 -19184.68} C_VEL
LIN {X 0,Y 244.357,Z 453.332,A -85,B 0,C 180,E1 -19187.145,E2 -19187.145} C_VEL
LIN {X 0,Y 246.353,Z 445.298,A -85,B 0,C 180,E1 -19189.509,E2 -19189.509} C_VEL
LIN {X 0,Y 248.267,Z 436.533,A -85,B 0,C 180,E1 -19191.592,E2 -19191.592} C_VEL
LIN {X 0,Y 250.673,Z 426.036,A -85,B 0,C 180,E1 -19193.547,E2 -19193.547} C_VEL
LIN {X 0,Y 251.204,Z 422.403,A -85,B 0,C 180,E1 -19194.151,E2 -19194.151} C_VEL
LIN {X 0,Y 250.877,Z 411.752,A -85,B 0,C 180,E1 -19195.851,E2 -19195.851} C_VEL
LIN {X 0,Y 249.881,Z 401.139,A -85,B 0,C 180,E1 -19197.308,E2 -19197.308} C_VEL
LIN {X 0,Y 247.905,Z 389.311,A -85,B 0,C 180,E1 -19198.723,E2 -19198.723} C_VEL
LIN {X 0,Y 244.7,Z 376.118,A -85,B 0,C 180,E1 -19200.087,E2 -19200.087} C_VEL
LIN {X 0,Y 242.836,Z 369.951,A -85,B 0,C 180,E1 -19200.652,E2 -19200.652} C_VEL
LIN {X 0,Y 242.824,Z 369.426,A -85,B 0,C 180,E1 -19200.738,E2 -19200.738} C_VEL
LIN {X 0,Y 243.634,Z 365.614,A -85,B 0,C 180,E1 -19204.228,E2 -19204.228} C_VEL
LIN {X 0,Y 243.937,Z 362.454,A -85,B 0,C 180,E1 -19207.229,E2 -19207.229} C_VEL
LIN {X 0,Y 243.856,Z 360.332,A -85,B 0,C 180,E1 -19209.347,E2 -19209.347} C_VEL
LIN {X 0,Y 243.409,Z 357.162,A -85,B 0,C 180,E1 -19212.671,E2 -19212.671} C_VEL
LIN {X 0,Y 242.761,Z 353.885,A -85,B 0,C 180,E1 -19216.363,E2 -19216.363} C_VEL
LIN {X 0,Y 242.186,Z 350.596,A -85,B 0,C 180,E1 -19220.326,E2 -19220.326} C_VEL
LIN {X 0,Y 241.982,Z 349.343,A -85,B 0,C 180,E1 -19222.019,E2 -19222.019} C_VEL
LIN {X 0,Y 241.973,Z 349.345,A -85,B 0,C 180,E1 -19226.506,E2 -19226.506} C_VEL
LIN {X 0,Y 241.971,Z 349.347,A -85,B 0,C 180,E1 -19230.612,E2 -19230.612} C_VEL
LIN {X 0,Y 242.026,Z 349.339,A -85,B 0,C 180,E1 -19234.178,E2 -19234.178} C_VEL
LIN {X 0,Y 242.019,Z 349.339,A -85,B 0,C 180,E1 -19238.313,E2 -19238.313} C_VEL
LIN {X 0,Y 242.157,Z 349.32,A -85,B 0,C 180,E1 -19243.278,E2 -19243.278} C_VEL
LIN {X 0,Y 242.179,Z 349.318,A -85,B 0,C 180,E1 -19248.279,E2 -19248.279} C_VEL
LIN {X 0,Y 242.421,Z 349.288,A -85,B 0,C 180,E1 -19251.665,E2 -19251.665} C_VEL
LIN {X 0,Y 242.255,Z 349.307,A -85,B 0,C 180,E1 -19255.007,E2 -19255.007} C_VEL
LIN {X 0,Y 242.628,Z 349.261,A -85,B 0,C 180,E1 -19258.34,E2 -19258.34} C_VEL
LIN {X 0,Y 242.627,Z 349.263,A -85,B 0,C 180,E1 -19261.66,E2 -19261.66} C_VEL
LIN {X 0,Y 242.424,Z 349.286,A -85,B 0,C 180,E1 -19266.71,E2 -19266.71} C_VEL
LIN {X 0,Y 242.339,Z 349.297,A -85,B 0,C 180,E1 -19270.021,E2 -19270.021} C_VEL
LIN {X 0,Y 242.16,Z 349.32,A -85,B 0,C 180,E1 -19275.141,E2 -19275.141} C_VEL
LIN {X 0,Y 242.066,Z 349.332,A -85,B 0,C 180,E1 -19278.625,E2 -19278.625} C_VEL
LIN {X 0,Y 241.999,Z 349.338,A -85,B 0,C 180,E1 -19282.181,E2 -19282.181} C_VEL
LIN {X 0,Y 242.026,Z 349.336,A -85,B 0,C 180,E1 -19285.822,E2 -19285.822} C_VEL
LIN {X 0,Y 241.963,Z 349.345,A -85,B 0,C 180,E1 -19289.589,E2 -19289.589} C_VEL
LIN {X 0,Y 241.974,Z 349.344,A -85,B 0,C 180,E1 -19293.494,E2 -19293.494} C_VEL
LIN {X 0,Y 241.982,Z 349.341,A -85,B 0,C 180,E1 -19297.584,E2 -19297.584} C_VEL
LIN {X 0,Y 241.908,Z 349.351,A -85,B 0,C 180,E1 -19301.929,E2 -19301.929} C_VEL
LIN {X 0,Y 241.936,Z 349.349,A -85,B 0,C 180,E1 -19306.571,E2 -19306.571} C_VEL
LIN {X 0,Y 241.961,Z 349.347,A -85,B 0,C 180,E1 -19308.085,E2 -19308.085} C_VEL
LIN {X 0,Y 242.284,Z 352.252,A -85,B 0,C 180,E1 -19312.473,E2 -19312.473} C_VEL
LIN {X 0,Y 242.289,Z 353.787,A -85,B 0,C 180,E1 -19314.542,E2 -19314.542} C_VEL
LIN {X 0,Y 241.869,Z 357.535,A -85,B 0,C 180,E1 -19319.245,E2 -19319.245} C_VEL
LIN {X 0,Y 244.003,Z 363.559,A -85,B 0,C 180,E1 -19319.882,E2 -19319.882} C_VEL
LIN {X 0,Y 247.67,Z 374.591,A -85,B 0,C 180,E1 -19321.159,E2 -19321.159} C_VEL
LIN {X 0,Y 250.636,Z 386.556,A -85,B 0,C 180,E1 -19322.706,E2 -19322.706} C_VEL
LIN {X 0,Y 252.562,Z 397.921,A -85,B 0,C 180,E1 -19324.373,E2 -19324.373} C_VEL
LIN {X 0,Y 253.138,Z 404.255,A -85,B 0,C 180,E1 -19325.39,E2 -19325.39} C_VEL
LIN {X 0,Y 250.898,Z 415.299,A -85,B 0,C 180,E1 -19327.152,E2 -19327.152} C_VEL
LIN {X 0,Y 249.094,Z 424.073,A -85,B 0,C 180,E1 -19328.917,E2 -19328.917} C_VEL
LIN {X 0,Y 246.81,Z 433.703,A -85,B 0,C 180,E1 -19331.317,E2 -19331.317} C_VEL
LIN {X 0,Y 244.707,Z 441.382,A -85,B 0,C 180,E1 -19333.74,E2 -19333.74} C_VEL
LIN {X 0,Y 243.388,Z 446.621,A -85,B 0,C 180,E1 -19335.793,E2 -19335.793} C_VEL
LIN {X 0,Y 242.046,Z 451.702,A -85,B 0,C 180,E1 -19338.274,E2 -19338.274} C_VEL
LIN {X 0,Y 241.066,Z 455.646,A -85,B 0,C 180,E1 -19340.774,E2 -19340.774} C_VEL
LIN {X 0,Y 240.426,Z 458.881,A -85,B 0,C 180,E1 -19343.656,E2 -19343.656} C_VEL
LIN {X 0,Y 240.046,Z 460.933,A -85,B 0,C 180,E1 -19346.644,E2 -19346.644} C_VEL
LIN {X 0,Y 239.947,Z 461.541,A -85,B 0,C 180,E1 -19348.322,E2 -19348.322} C_VEL
LIN {X 0,Y 239.927,Z 461.769,A -85,B 0,C 180,E1 -19350.001,E2 -19350.001} C_VEL
LIN {X 0,Y 239.947,Z 461.575,A -85,B 0,C 180,E1 -19351.679,E2 -19351.679} C_VEL
LIN {X 0,Y 240.039,Z 460.989,A -85,B 0,C 180,E1 -19353.358,E2 -19353.358} C_VEL
LIN {X 0,Y 240.49,Z 458.666,A -85,B 0,C 180,E1 -19356.714,E2 -19356.714} C_VEL
LIN {X 0,Y 241.095,Z 455.8,A -85,B 0,C 180,E1 -19359.226,E2 -19359.226} C_VEL
LIN {X 0,Y 241.99,Z 451.913,A -85,B 0,C 180,E1 -19361.73,E2 -19361.73} C_VEL
LIN {X 0,Y 243.32,Z 446.893,A -85,B 0,C 180,E1 -19364.213,E2 -19364.213} C_VEL
LIN {X 0,Y 244.951,Z 440.571,A -85,B 0,C 180,E1 -19366.674,E2 -19366.674} C_VEL
LIN {X 0,Y 247.071,Z 432.655,A -85,B 0,C 180,E1 -19369.094,E2 -19369.094} C_VEL
LIN {X 0,Y 249.114,Z 424.128,A -85,B 0,C 180,E1 -19371.194,E2 -19371.194} C_VEL
LIN {X 0,Y 251.094,Z 414.742,A -85,B 0,C 180,E1 -19373.07,E2 -19373.07} C_VEL
LIN {X 0,Y 253.202,Z 403.98,A -85,B 0,C 180,E1 -19374.773,E2 -19374.773} C_VEL
LIN {X 0,Y 251.875,Z 392.881,A -85,B 0,C 180,E1 -19376.516,E2 -19376.516} C_VEL
LIN {X 0,Y 249.531,Z 381.536,A -85,B 0,C 180,E1 -19378.093,E2 -19378.093} C_VEL
LIN {X 0,Y 246.146,Z 369.64,A -85,B 0,C 180,E1 -19379.56,E2 -19379.56} C_VEL
LIN {X 0,Y 241.934,Z 357.961,A -85,B 0,C 180,E1 -19380.839,E2 -19380.839} C_VEL
LIN {X 0,Y 241.866,Z 357.501,A -85,B 0,C 180,E1 -19380.939,E2 -19380.939} C_VEL
LIN {X 0,Y 242.268,Z 353.897,A -85,B 0,C 180,E1 -19385.464,E2 -19385.464} C_VEL
LIN {X 0,Y 242.254,Z 351.72,A -85,B 0,C 180,E1 -19388.437,E2 -19388.437} C_VEL
LIN {X 0,Y 241.956,Z 349.35,A -85,B 0,C 180,E1 -19391.918,E2 -19391.918} C_VEL
LIN {X 0,Y 241.909,Z 349.354,A -85,B 0,C 180,E1 -19396.578,E2 -19396.578} C_VEL
LIN {X 0,Y 241.984,Z 349.343,A -85,B 0,C 180,E1 -19401.643,E2 -19401.643} C_VEL
LIN {X 0,Y 241.974,Z 349.343,A -85,B 0,C 180,E1 -19404.487,E2 -19404.487} C_VEL
LIN {X 0,Y 241.952,Z 349.343,A -85,B 0,C 180,E1 -19408.476,E2 -19408.476} C_VEL
LIN {X 0,Y 241.967,Z 349.343,A -85,B 0,C 180,E1 -19412.307,E2 -19412.307} C_VEL
LIN {X 0,Y 242.024,Z 349.335,A -85,B 0,C 180,E1 -19416.012,E2 -19416.012} C_VEL
LIN {X 0,Y 242.035,Z 349.335,A -85,B 0,C 180,E1 -19419.608,E2 -19419.608} C_VEL
LIN {X 0,Y 242.163,Z 349.32,A -85,B 0,C 180,E1 -19423.278,E2 -19423.278} C_VEL
LIN {X 0,Y 242.185,Z 349.316,A -85,B 0,C 180,E1 -19428.28,E2 -19428.28} C_VEL
LIN {X 0,Y 242.427,Z 349.286,A -85,B 0,C 180,E1 -19431.665,E2 -19431.665} C_VEL
LIN {X 0,Y 242.257,Z 349.307,A -85,B 0,C 180,E1 -19435.007,E2 -19435.007} C_VEL
LIN {X 0,Y 242.632,Z 349.262,A -85,B 0,C 180,E1 -19438.34,E2 -19438.34} C_VEL
LIN {X 0,Y 242.632,Z 349.26,A -85,B 0,C 180,E1 -19441.66,E2 -19441.66} C_VEL
LIN {X 0,Y 242.422,Z 349.289,A -85,B 0,C 180,E1 -19446.659,E2 -19446.659} C_VEL
LIN {X 0,Y 242.267,Z 349.311,A -85,B 0,C 180,E1 -19450.024,E2 -19450.024} C_VEL
LIN {X 0,Y 242.163,Z 349.321,A -85,B 0,C 180,E1 -19455.141,E2 -19455.141} C_VEL
LIN {X 0,Y 242.071,Z 349.332,A -85,B 0,C 180,E1 -19458.624,E2 -19458.624} C_VEL
LIN {X 0,Y 242.004,Z 349.34,A -85,B 0,C 180,E1 -19462.181,E2 -19462.181} C_VEL
LIN {X 0,Y 242.032,Z 349.337,A -85,B 0,C 180,E1 -19465.821,E2 -19465.821} C_VEL
LIN {X 0,Y 241.968,Z 349.347,A -85,B 0,C 180,E1 -19469.589,E2 -19469.589} C_VEL
LIN {X 0,Y 241.978,Z 349.346,A -85,B 0,C 180,E1 -19473.493,E2 -19473.493} C_VEL
LIN {X 0,Y 241.99,Z 349.39,A -85,B 0,C 180,E1 -19478.098,E2 -19478.098} C_VEL
LIN {X 0,Y 242.434,Z 352.4,A -85,B 0,C 180,E1 -19481.817,E2 -19481.817} C_VEL
LIN {X 0,Y 242.721,Z 353.957,A -85,B 0,C 180,E1 -19483.658,E2 -19483.658} C_VEL
LIN {X 0,Y 242.29,Z 355.265,A -85,B 0,C 180,E1 -19485.013,E2 -19485.013} C_VEL
LIN {X 0,Y 239.869,Z 357.734,A -85,B 0,C 180,E1 -19487.22,E2 -19487.22} C_VEL
LIN {X 0,Y 237.039,Z 360.771,A -85,B 0,C 180,E1 -19489.93,E2 -19489.93} C_VEL
LIN {X 0,Y 236.789,Z 361.71,A -85,B 0,C 180,E1 -19490.867,E2 -19490.867} C_VEL
LIN {X 0,Y 236.813,Z 364.377,A -85,B 0,C 180,E1 -19493.591,E2 -19493.591} C_VEL
LIN {X 0,Y 236.444,Z 367.178,A -85,B 0,C 180,E1 -19496.332,E2 -19496.332} C_VEL
LIN {X 0,Y 235.974,Z 369.248,A -85,B 0,C 180,E1 -19498.275,E2 -19498.275} C_VEL
LIN {X 0,Y 238.59,Z 378.478,A -85,B 0,C 180,E1 -19499.187,E2 -19499.187} C_VEL
LIN {X 0,Y 241.525,Z 390.874,A -85,B 0,C 180,E1 -19500.57,E2 -19500.57} C_VEL
LIN {X 0,Y 243.484,Z 402.917,A -85,B 0,C 180,E1 -19502.11,E2 -19502.11} C_VEL
LIN {X 0,Y 244.385,Z 413.893,A -85,B 0,C 180,E1 -19503.722,E2 -19503.722} C_VEL
LIN {X 0,Y 244.554,Z 423.621,A -85,B 0,C 180,E1 -19505.373,E2 -19505.373} C_VEL
LIN {X 0,Y 242.636,Z 432.541,A -85,B 0,C 180,E1 -19506.981,E2 -19506.981} C_VEL
LIN {X 0,Y 240.454,Z 441.704,A -85,B 0,C 180,E1 -19509.02,E2 -19509.02} C_VEL
LIN {X 0,Y 238.215,Z 450.639,A -85,B 0,C 180,E1 -19511.509,E2 -19511.509} C_VEL
LIN {X 0,Y 236.307,Z 457.83,A -85,B 0,C 180,E1 -19514.031,E2 -19514.031} C_VEL
LIN {X 0,Y 234.995,Z 462.685,A -85,B 0,C 180,E1 -19516.157,E2 -19516.157} C_VEL
LIN {X 0,Y 233.952,Z 467.411,A -85,B 0,C 180,E1 -19518.739,E2 -19518.739} C_VEL
LIN {X 0,Y 233.241,Z 471.024,A -85,B 0,C 180,E1 -19521.334,E2 -19521.334} C_VEL
LIN {X 0,Y 232.927,Z 472.888,A -85,B 0,C 180,E1 -19523.067,E2 -19523.067} C_VEL
LIN {X 0,Y 232.755,Z 474.522,A -85,B 0,C 180,E1 -19525.159,E2 -19525.159} C_VEL
LIN {X 0,Y 232.748,Z 475.9,A -85,B 0,C 180,E1 -19528.269,E2 -19528.269} C_VEL
LIN {X 0,Y 232.784,Z 476.116,A -85,B 0,C 180,E1 -19529.999,E2 -19529.999} C_VEL
LIN {X 0,Y 232.748,Z 475.893,A -85,B 0,C 180,E1 -19531.73,E2 -19531.73} C_VEL
LIN {X 0,Y 232.767,Z 474.272,A -85,B 0,C 180,E1 -19535.196,E2 -19535.196} C_VEL
LIN {X 0,Y 232.926,Z 472.865,A -85,B 0,C 180,E1 -19536.931,E2 -19536.931} C_VEL
LIN {X 0,Y 233.441,Z 469.915,A -85,B 0,C 180,E1 -19539.53,E2 -19539.53} C_VEL
LIN {X 0,Y 234.283,Z 465.927,A -85,B 0,C 180,E1 -19542.12,E2 -19542.12} C_VEL
LIN {X 0,Y 235.767,Z 459.799,A -85,B 0,C 180,E1 -19545.118,E2 -19545.118} C_VEL
LIN {X 0,Y 237.52,Z 453.112,A -85,B 0,C 180,E1 -19547.654,E2 -19547.654} C_VEL
LIN {X 0,Y 239.465,Z 445.762,A -85,B 0,C 180,E1 -19549.889,E2 -19549.889} C_VEL
LIN {X 0,Y 241.658,Z 436.314,A -85,B 0,C 180,E1 -19552.213,E2 -19552.213} C_VEL
LIN {X 0,Y 243.901,Z 426.992,A -85,B 0,C 180,E1 -19554.016,E2 -19554.016} C_VEL
LIN {X 0,Y 244.492,Z 423.453,A -85,B 0,C 180,E1 -19554.632,E2 -19554.632} C_VEL
LIN {X 0,Y 244.325,Z 413.828,A -85,B 0,C 180,E1 -19556.261,E2 -19556.261} C_VEL
LIN {X 0,Y 243.423,Z 402.735,A -85,B 0,C 180,E1 -19557.883,E2 -19557.883} C_VEL
LIN {X 0,Y 241.467,Z 390.807,A -85,B 0,C 180,E1 -19559.405,E2 -19559.405} C_VEL
LIN {X 0,Y 238.541,Z 378.277,A -85,B 0,C 180,E1 -19560.793,E2 -19560.793} C_VEL
LIN {X 0,Y 236.03,Z 369.891,A -85,B 0,C 180,E1 -19561.628,E2 -19561.628} C_VEL
LIN {X 0,Y 235.965,Z 369.211,A -85,B 0,C 180,E1 -19561.723,E2 -19561.723} C_VEL
LIN {X 0,Y 236.732,Z 365.379,A -85,B 0,C 180,E1 -19565.372,E2 -19565.372} C_VEL
LIN {X 0,Y 236.87,Z 362.22,A -85,B 0,C 180,E1 -19568.539,E2 -19568.539} C_VEL
LIN {X 0,Y 236.522,Z 358.959,A -85,B 0,C 180,E1 -19572.025,E2 -19572.025} C_VEL
LIN {X 0,Y 235.711,Z 354.903,A -85,B 0,C 180,E1 -19576.704,E2 -19576.704} C_VEL
LIN {X 0,Y 235.119,Z 351.38,A -85,B 0,C 180,E1 -19581.118,E2 -19581.118} C_VEL
LIN {X 0,Y 234.913,Z 350.222,A -85,B 0,C 180,E1 -19582.712,E2 -19582.712} C_VEL
LIN {X 0,Y 234.947,Z 350.221,A -85,B 0,C 180,E1 -19587.423,E2 -19587.423} C_VEL
LIN {X 0,Y 234.895,Z 350.227,A -85,B 0,C 180,E1 -19591.398,E2 -19591.398} C_VEL
LIN {X 0,Y 234.948,Z 350.22,A -85,B 0,C 180,E1 -19595.242,E2 -19595.242} C_VEL
LIN {X 0,Y 234.991,Z 350.213,A -85,B 0,C 180,E1 -19598.968,E2 -19598.968} C_VEL
LIN {X 0,Y 235.09,Z 350.201,A -85,B 0,C 180,E1 -19603.059,E2 -19603.059} C_VEL
LIN {X 0,Y 235.139,Z 350.197,A -85,B 0,C 180,E1 -19607.923,E2 -19607.923} C_VEL
LIN {X 0,Y 235.37,Z 350.166,A -85,B 0,C 180,E1 -19611.414,E2 -19611.414} C_VEL
LIN {X 0,Y 235.398,Z 350.162,A -85,B 0,C 180,E1 -19613.141,E2 -19613.141} C_VEL
LIN {X 0,Y 235.588,Z 350.139,A -85,B 0,C 180,E1 -19618.291,E2 -19618.291} C_VEL
LIN {X 0,Y 235.587,Z 350.139,A -85,B 0,C 180,E1 -19621.71,E2 -19621.71} C_VEL
LIN {X 0,Y 235.399,Z 350.162,A -85,B 0,C 180,E1 -19626.859,E2 -19626.859} C_VEL
LIN {X 0,Y 235.247,Z 350.18,A -85,B 0,C 180,E1 -19630.326,E2 -19630.326} C_VEL
LIN {X 0,Y 235.107,Z 350.199,A -85,B 0,C 180,E1 -19635.607,E2 -19635.607} C_VEL
LIN {X 0,Y 235.002,Z 350.212,A -85,B 0,C 180,E1 -19639.206,E2 -19639.206} C_VEL
LIN {X 0,Y 234.941,Z 350.22,A -85,B 0,C 180,E1 -19642.885,E2 -19642.885} C_VEL
LIN {X 0,Y 234.939,Z 350.22,A -85,B 0,C 180,E1 -19646.661,E2 -19646.661} C_VEL
LIN {X 0,Y 234.893,Z 350.227,A -85,B 0,C 180,E1 -19650.574,E2 -19650.574} C_VEL
LIN {X 0,Y 234.924,Z 350.223,A -85,B 0,C 180,E1 -19654.639,E2 -19654.639} C_VEL
LIN {X 0,Y 234.907,Z 350.225,A -85,B 0,C 180,E1 -19658.936,E2 -19658.936} C_VEL
LIN {X 0,Y 234.876,Z 350.228,A -85,B 0,C 180,E1 -19664.102,E2 -19664.102} C_VEL
LIN {X 0,Y 234.913,Z 350.224,A -85,B 0,C 180,E1 -19666.522,E2 -19666.522} C_VEL
LIN {X 0,Y 235.01,Z 350.968,A -85,B 0,C 180,E1 -19668.861,E2 -19668.861} C_VEL
LIN {X 0,Y 235.191,Z 352.488,A -85,B 0,C 180,E1 -19671.134,E2 -19671.134} C_VEL
LIN {X 0,Y 235.272,Z 354.343,A -85,B 0,C 180,E1 -19673.759,E2 -19673.759} C_VEL
LIN {X 0,Y 234.969,Z 357.938,A -85,B 0,C 180,E1 -19678.27,E2 -19678.27} C_VEL
LIN {X 0,Y 236.023,Z 361.026,A -85,B 0,C 180,E1 -19678.594,E2 -19678.594} C_VEL
LIN {X 0,Y 240.357,Z 373.044,A -85,B 0,C 180,E1 -19680.047,E2 -19680.047} C_VEL
LIN {X 0,Y 243.532,Z 384.927,A -85,B 0,C 180,E1 -19681.621,E2 -19681.621} C_VEL
LIN {X 0,Y 245.672,Z 396.834,A -85,B 0,C 180,E1 -19683.406,E2 -19683.406} C_VEL
LIN {X 0,Y 246.472,Z 405.813,A -85,B 0,C 180,E1 -19684.904,E2 -19684.904} C_VEL
LIN {X 0,Y 244.135,Z 416.689,A -85,B 0,C 180,E1 -19686.729,E2 -19686.729} C_VEL
LIN {X 0,Y 242.086,Z 426.14,A -85,B 0,C 180,E1 -19688.743,E2 -19688.743} C_VEL
LIN {X 0,Y 240.101,Z 433.921,A -85,B 0,C 180,E1 -19690.775,E2 -19690.775} C_VEL
LIN {X 0,Y 237.898,Z 441.6,A -85,B 0,C 180,E1 -19693.261,E2 -19693.261} C_VEL
LIN {X 0,Y 236.508,Z 446.839,A -85,B 0,C 180,E1 -19695.371,E2 -19695.371} C_VEL
LIN {X 0,Y 235.089,Z 451.919,A -85,B 0,C 180,E1 -19697.922,E2 -19697.922} C_VEL
LIN {X 0,Y 234.054,Z 455.862,A -85,B 0,C 180,E1 -19700.495,E2 -19700.495} C_VEL
LIN {X 0,Y 233.314,Z 459.332,A -85,B 0,C 180,E1 -19703.746,E2 -19703.746} C_VEL
